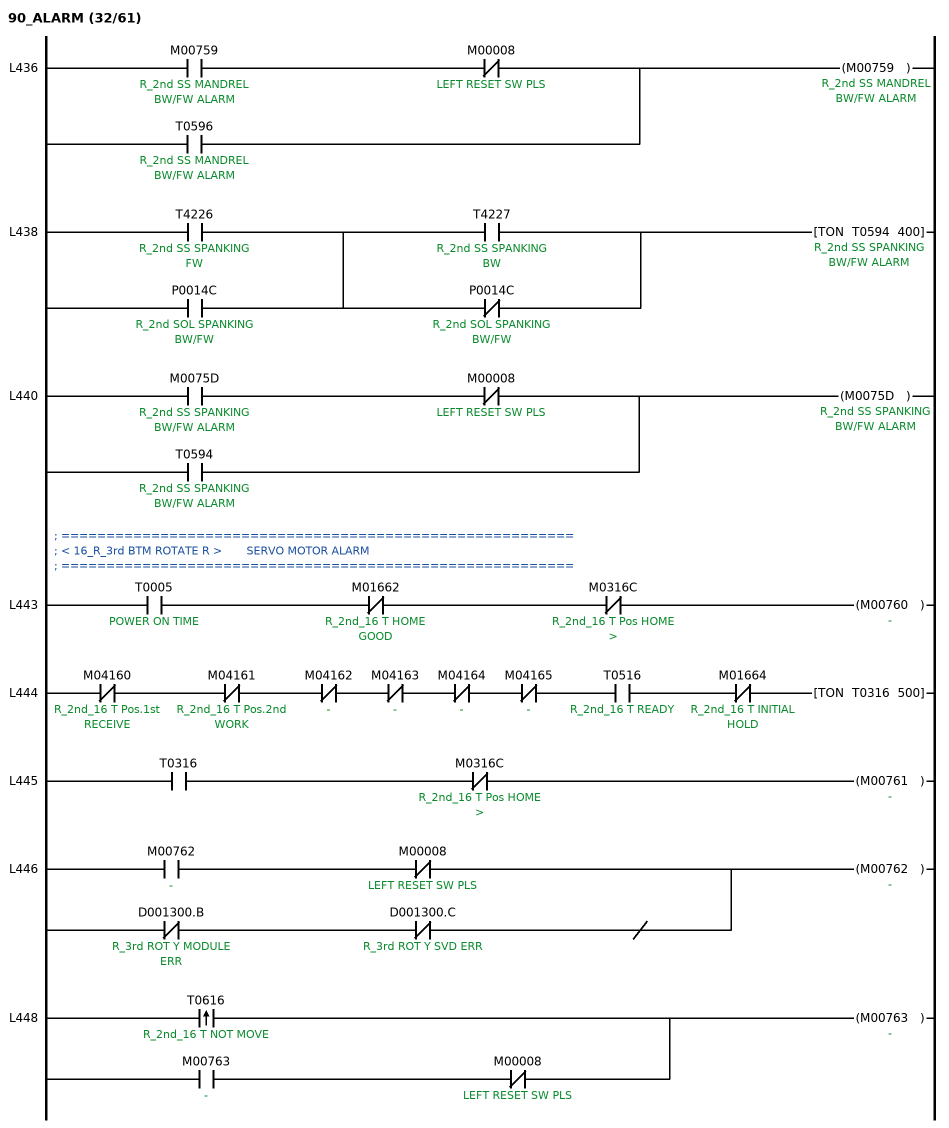
[picture p408: 90_ALARM rungs L436-L448]
; L436
LOAD      M00759	// R_2nd SS MANDREL BW/FW ALARM
AND NOT   M00008	// LEFT RESET SW PLS
OR        T0596	// R_2nd SS MANDREL BW/FW ALARM
OUT       M00759	// R_2nd SS MANDREL BW/FW ALARM
; L438
LOAD      T4226	// R_2nd SS SPANKING FW
OR        P0014C	// R_2nd SOL SPANKING BW/FW
LOAD      T4227	// R_2nd SS SPANKING BW
OR NOT    P0014C	// R_2nd SOL SPANKING BW/FW
AND LOAD
TON       T0594 400	// R_2nd SS SPANKING BW/FW ALARM
; L440
LOAD      M0075D	// R_2nd SS SPANKING BW/FW ALARM
AND NOT   M00008	// LEFT RESET SW PLS
OR        T0594	// R_2nd SS SPANKING BW/FW ALARM
OUT       M0075D	// R_2nd SS SPANKING BW/FW ALARM
// =========================================================
// 
//        < 16_R_3rd BTM ROTATE R >       SERVO MOTOR ALARM
// 
// =========================================================
; L443
LOAD      T0005	// POWER ON TIME
AND NOT   M01662	// R_2nd_16 T HOME GOOD
AND NOT   M0316C	// R_2nd_16 T Pos HOME >
OUT       M00760	// -
; L444
LOAD NOT  M04160	// R_2nd_16 T Pos.1st RECEIVE
AND NOT   M04161	// R_2nd_16 T Pos.2nd WORK
AND NOT   M04162	// -
AND NOT   M04163	// -
AND NOT   M04164	// -
AND NOT   M04165	// -
AND       T0516	// R_2nd_16 T READY
AND NOT   M01664	// R_2nd_16 T INITIAL HOLD
TON       T0316 500
; L445
LOAD      T0316
AND NOT   M0316C	// R_2nd_16 T Pos HOME >
OUT       M00761	// -
; L446
LOAD      M00762	// -
AND NOT   M00008	// LEFT RESET SW PLS
LOAD NOT  D001300.B	// R_3rd ROT Y MODULE ERR
AND NOT   D001300.C	// R_3rd ROT Y SVD ERR
NOT
OR LOAD
OUT       M00762	// -
; L448
LOADP     T0616	// R_2nd_16 T NOT MOVE
LOAD      M00763	// -
AND NOT   M00008	// LEFT RESET SW PLS
OR LOAD
OUT       M00763	// -

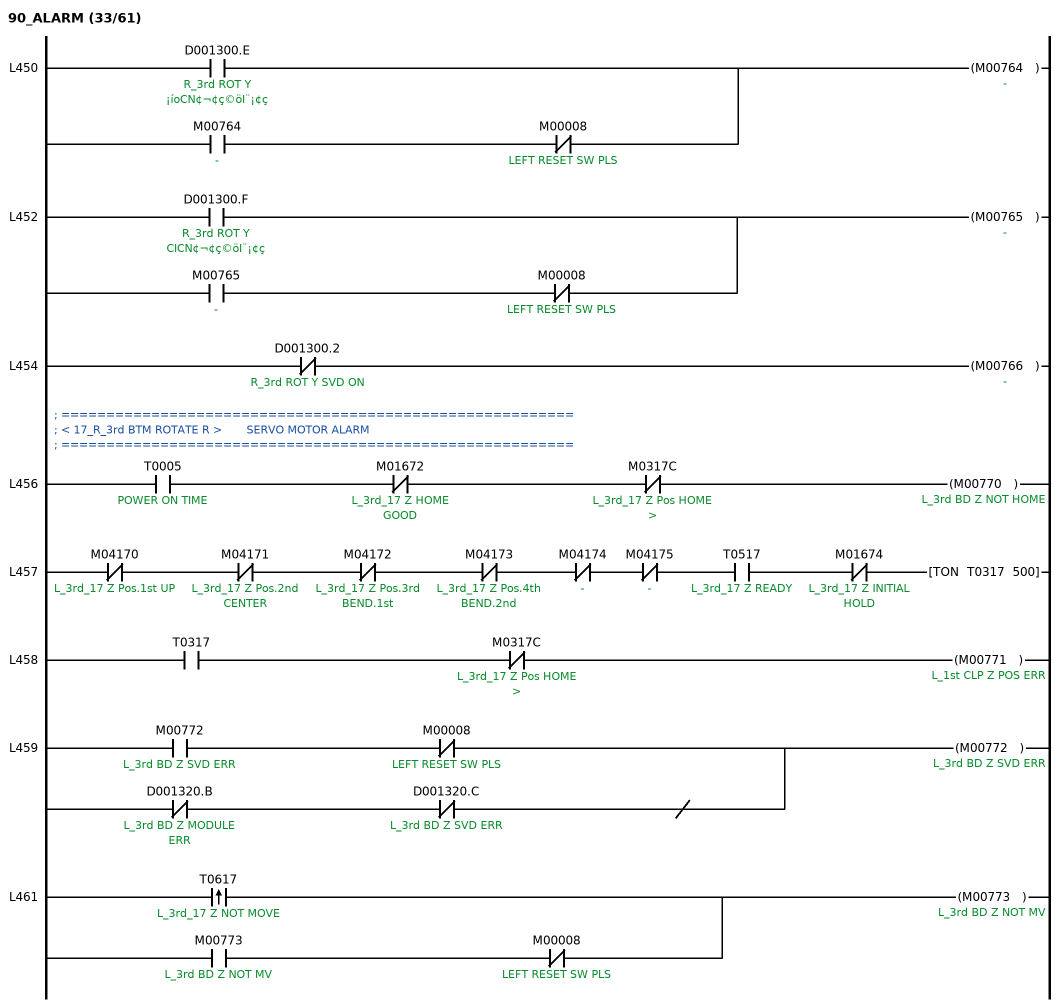
; L450
LOAD      D001300.E	// R_3rd ROT Y ¡íoCN¢¬¢ç©öI¨¡¢ç
LOAD      M00764	// -
AND NOT   M00008	// LEFT RESET SW PLS
OR LOAD
OUT       M00764	// -
; L452
LOAD      D001300.F	// R_3rd ROT Y CICN¢¬¢ç©öI¨¡¢ç
LOAD      M00765	// -
AND NOT   M00008	// LEFT RESET SW PLS
OR LOAD
OUT       M00765	// -
; L454
LOAD NOT  D001300.2	// R_3rd ROT Y SVD ON
OUT       M00766	// -
// =========================================================
// 
//        < 17_R_3rd BTM ROTATE R >       SERVO MOTOR ALARM
// 
// =========================================================
; L456
LOAD      T0005	// POWER ON TIME
AND NOT   M01672	// L_3rd_17 Z HOME GOOD
AND NOT   M0317C	// L_3rd_17 Z Pos HOME >
OUT       M00770	// L_3rd BD Z NOT HOME
; L457
LOAD NOT  M04170	// L_3rd_17 Z Pos.1st UP
AND NOT   M04171	// L_3rd_17 Z Pos.2nd CENTER
AND NOT   M04172	// L_3rd_17 Z Pos.3rd BEND.1st
AND NOT   M04173	// L_3rd_17 Z Pos.4th BEND.2nd
AND NOT   M04174	// -
AND NOT   M04175	// -
AND       T0517	// L_3rd_17 Z READY
AND NOT   M01674	// L_3rd_17 Z INITIAL HOLD
TON       T0317 500
; L458
LOAD      T0317
AND NOT   M0317C	// L_3rd_17 Z Pos HOME >
OUT       M00771	// L_1st CLP Z POS ERR
; L459
LOAD      M00772	// L_3rd BD Z SVD ERR
AND NOT   M00008	// LEFT RESET SW PLS
LOAD NOT  D001320.B	// L_3rd BD Z MODULE ERR
AND NOT   D001320.C	// L_3rd BD Z SVD ERR
NOT
OR LOAD
OUT       M00772	// L_3rd BD Z SVD ERR
; L461
LOADP     T0617	// L_3rd_17 Z NOT MOVE
LOAD      M00773	// L_3rd BD Z NOT MV
AND NOT   M00008	// LEFT RESET SW PLS
OR LOAD
OUT       M00773	// L_3rd BD Z NOT MV

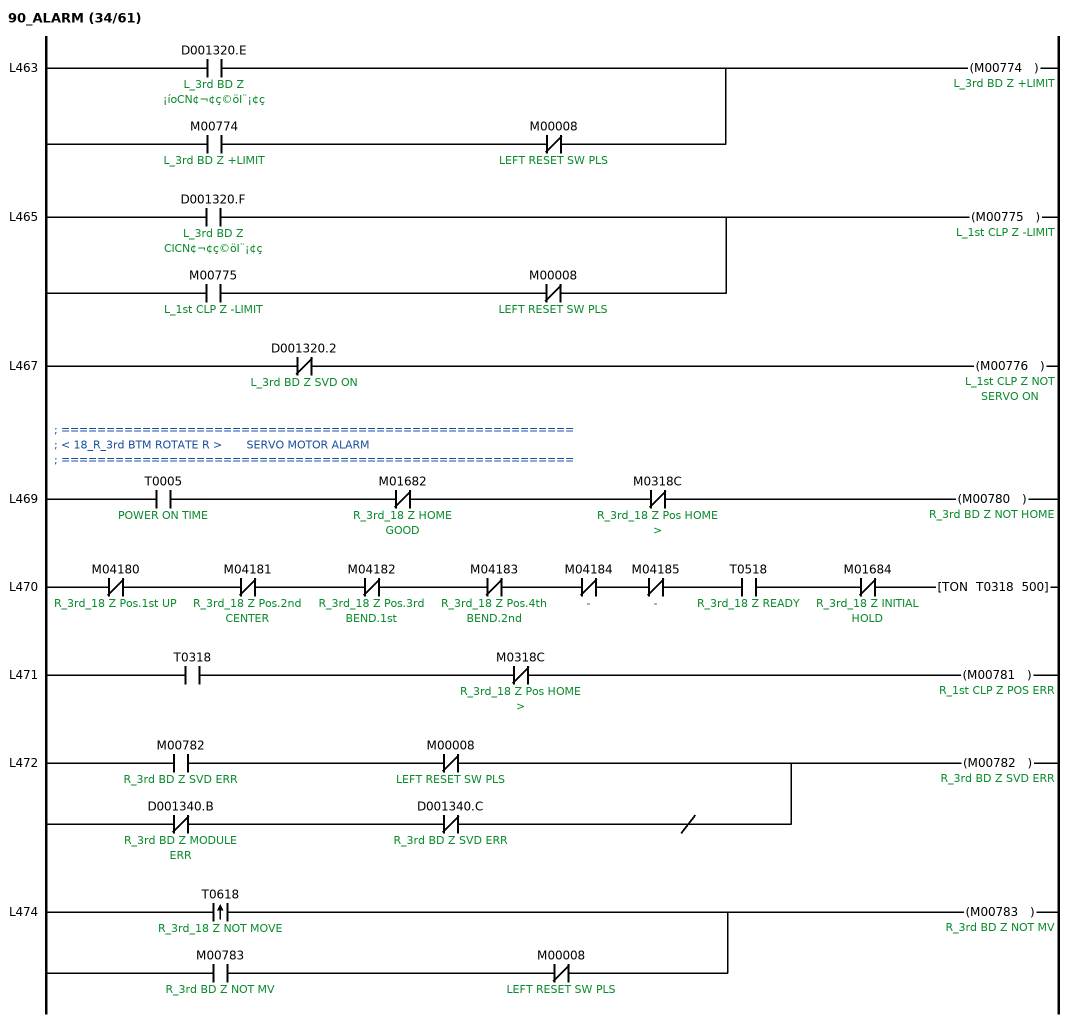
; L463
LOAD      D001320.E	// L_3rd BD Z ¡íoCN¢¬¢ç©öI¨¡¢ç
LOAD      M00774	// L_3rd BD Z +LIMIT
AND NOT   M00008	// LEFT RESET SW PLS
OR LOAD
OUT       M00774	// L_3rd BD Z +LIMIT
; L465
LOAD      D001320.F	// L_3rd BD Z CICN¢¬¢ç©öI¨¡¢ç
LOAD      M00775	// L_1st CLP Z -LIMIT
AND NOT   M00008	// LEFT RESET SW PLS
OR LOAD
OUT       M00775	// L_1st CLP Z -LIMIT
; L467
LOAD NOT  D001320.2	// L_3rd BD Z SVD ON
OUT       M00776	// L_1st CLP Z NOT SERVO ON
// =========================================================
// 
//        < 18_R_3rd BTM ROTATE R >       SERVO MOTOR ALARM
// 
// =========================================================
; L469
LOAD      T0005	// POWER ON TIME
AND NOT   M01682	// R_3rd_18 Z HOME GOOD
AND NOT   M0318C	// R_3rd_18 Z Pos HOME >
OUT       M00780	// R_3rd BD Z NOT HOME
; L470
LOAD NOT  M04180	// R_3rd_18 Z Pos.1st UP
AND NOT   M04181	// R_3rd_18 Z Pos.2nd CENTER
AND NOT   M04182	// R_3rd_18 Z Pos.3rd BEND.1st
AND NOT   M04183	// R_3rd_18 Z Pos.4th BEND.2nd
AND NOT   M04184	// -
AND NOT   M04185	// -
AND       T0518	// R_3rd_18 Z READY
AND NOT   M01684	// R_3rd_18 Z INITIAL HOLD
TON       T0318 500
; L471
LOAD      T0318
AND NOT   M0318C	// R_3rd_18 Z Pos HOME >
OUT       M00781	// R_1st CLP Z POS ERR
; L472
LOAD      M00782	// R_3rd BD Z SVD ERR
AND NOT   M00008	// LEFT RESET SW PLS
LOAD NOT  D001340.B	// R_3rd BD Z MODULE ERR
AND NOT   D001340.C	// R_3rd BD Z SVD ERR
NOT
OR LOAD
OUT       M00782	// R_3rd BD Z SVD ERR
; L474
LOADP     T0618	// R_3rd_18 Z NOT MOVE
LOAD      M00783	// R_3rd BD Z NOT MV
AND NOT   M00008	// LEFT RESET SW PLS
OR LOAD
OUT       M00783	// R_3rd BD Z NOT MV

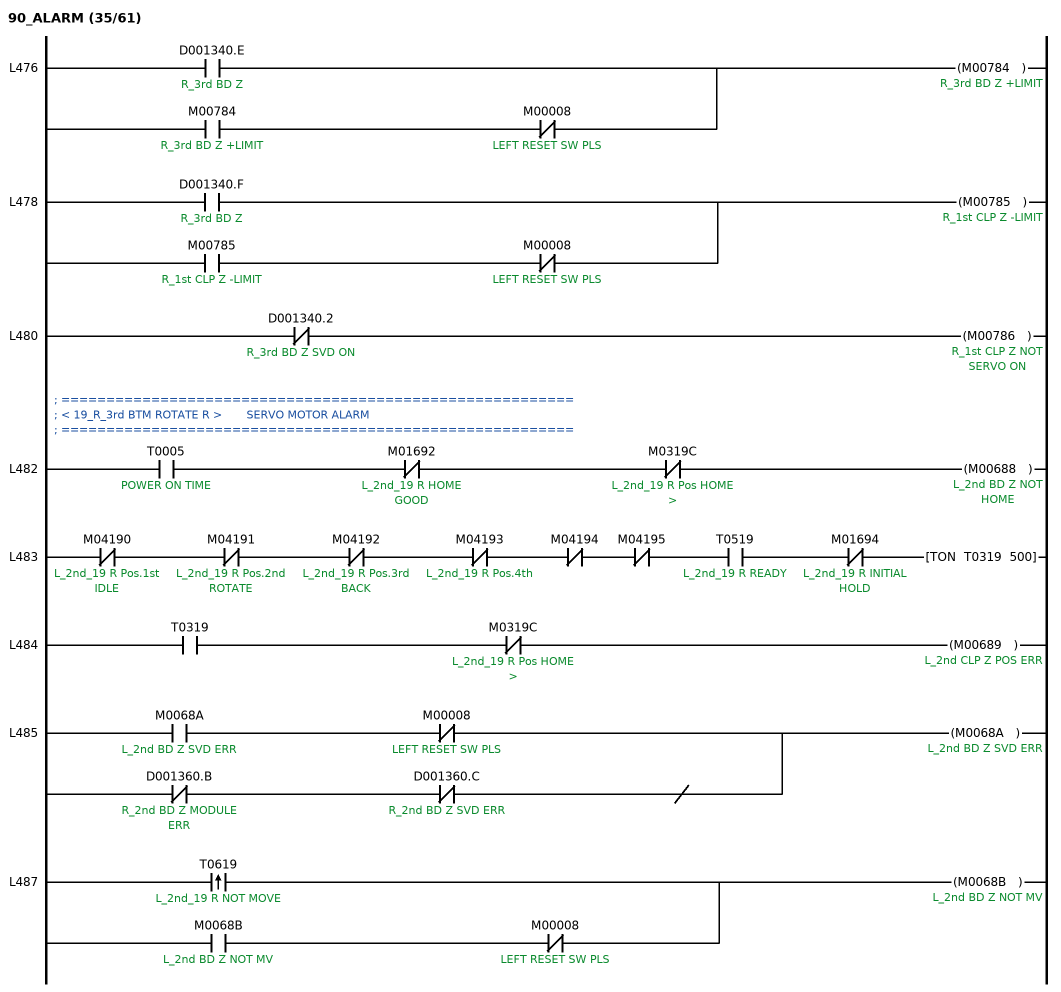
; L476
LOAD      D001340.E	// R_3rd BD Z
LOAD      M00784	// R_3rd BD Z +LIMIT
AND NOT   M00008	// LEFT RESET SW PLS
OR LOAD
OUT       M00784	// R_3rd BD Z +LIMIT
; L478
LOAD      D001340.F	// R_3rd BD Z
LOAD      M00785	// R_1st CLP Z -LIMIT
AND NOT   M00008	// LEFT RESET SW PLS
OR LOAD
OUT       M00785	// R_1st CLP Z -LIMIT
; L480
LOAD NOT  D001340.2	// R_3rd BD Z SVD ON
OUT       M00786	// R_1st CLP Z NOT SERVO ON
// =========================================================
// 
//        < 19_R_3rd BTM ROTATE R >       SERVO MOTOR ALARM
// 
// =========================================================
; L482
LOAD      T0005	// POWER ON TIME
AND NOT   M01692	// L_2nd_19 R HOME GOOD
AND NOT   M0319C	// L_2nd_19 R Pos HOME >
OUT       M00688	// L_2nd BD Z NOT HOME
; L483
LOAD NOT  M04190	// L_2nd_19 R Pos.1st IDLE
AND NOT   M04191	// L_2nd_19 R Pos.2nd ROTATE
AND NOT   M04192	// L_2nd_19 R Pos.3rd BACK
AND NOT   M04193	// L_2nd_19 R Pos.4th 
AND NOT   M04194
AND NOT   M04195
AND       T0519	// L_2nd_19 R READY
AND NOT   M01694	// L_2nd_19 R INITIAL HOLD
TON       T0319 500
; L484
LOAD      T0319
AND NOT   M0319C	// L_2nd_19 R Pos HOME >
OUT       M00689	// L_2nd CLP Z POS ERR
; L485
LOAD      M0068A	// L_2nd BD Z SVD ERR
AND NOT   M00008	// LEFT RESET SW PLS
LOAD NOT  D001360.B	// R_2nd BD Z MODULE ERR
AND NOT   D001360.C	// R_2nd BD Z SVD ERR
NOT
OR LOAD
OUT       M0068A	// L_2nd BD Z SVD ERR
; L487
LOADP     T0619	// L_2nd_19 R NOT MOVE
LOAD      M0068B	// L_2nd BD Z NOT MV
AND NOT   M00008	// LEFT RESET SW PLS
OR LOAD
OUT       M0068B	// L_2nd BD Z NOT MV

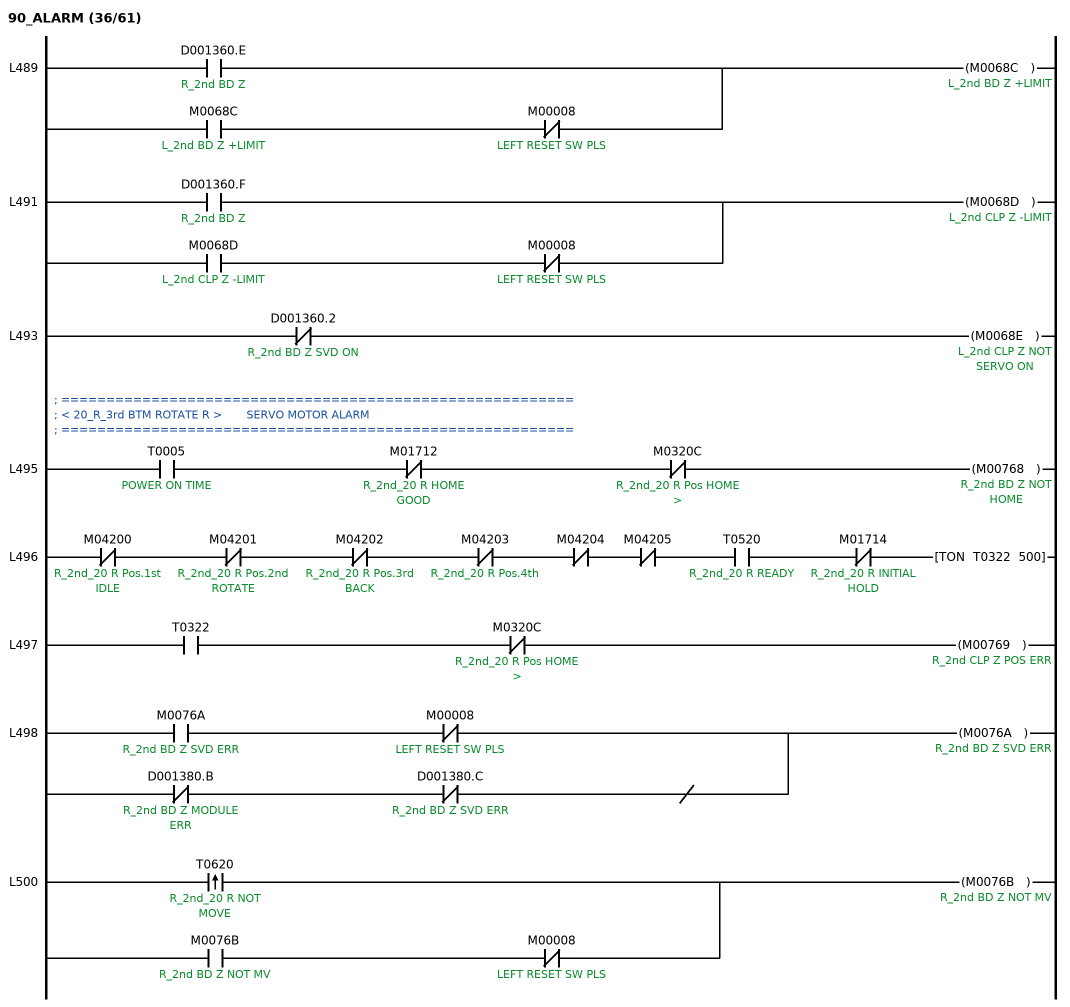
; L489
LOAD      D001360.E	// R_2nd BD Z
LOAD      M0068C	// L_2nd BD Z +LIMIT
AND NOT   M00008	// LEFT RESET SW PLS
OR LOAD
OUT       M0068C	// L_2nd BD Z +LIMIT
; L491
LOAD      D001360.F	// R_2nd BD Z
LOAD      M0068D	// L_2nd CLP Z -LIMIT
AND NOT   M00008	// LEFT RESET SW PLS
OR LOAD
OUT       M0068D	// L_2nd CLP Z -LIMIT
; L493
LOAD NOT  D001360.2	// R_2nd BD Z SVD ON
OUT       M0068E	// L_2nd CLP Z NOT SERVO ON
// =========================================================
// 
//        < 20_R_3rd BTM ROTATE R >       SERVO MOTOR ALARM
// 
// =========================================================
; L495
LOAD      T0005	// POWER ON TIME
AND NOT   M01712	// R_2nd_20 R HOME GOOD
AND NOT   M0320C	// R_2nd_20 R Pos HOME >
OUT       M00768	// R_2nd BD Z NOT HOME
; L496
LOAD NOT  M04200	// R_2nd_20 R Pos.1st IDLE
AND NOT   M04201	// R_2nd_20 R Pos.2nd ROTATE
AND NOT   M04202	// R_2nd_20 R Pos.3rd BACK
AND NOT   M04203	// R_2nd_20 R Pos.4th 
AND NOT   M04204
AND NOT   M04205
AND       T0520	// R_2nd_20 R READY
AND NOT   M01714	// R_2nd_20 R INITIAL HOLD
TON       T0322 500
; L497
LOAD      T0322
AND NOT   M0320C	// R_2nd_20 R Pos HOME >
OUT       M00769	// R_2nd CLP Z POS ERR
; L498
LOAD      M0076A	// R_2nd BD Z SVD ERR
AND NOT   M00008	// LEFT RESET SW PLS
LOAD NOT  D001380.B	// R_2nd BD Z MODULE ERR
AND NOT   D001380.C	// R_2nd BD Z SVD ERR
NOT
OR LOAD
OUT       M0076A	// R_2nd BD Z SVD ERR
; L500
LOADP     T0620	// R_2nd_20 R NOT MOVE
LOAD      M0076B	// R_2nd BD Z NOT MV
AND NOT   M00008	// LEFT RESET SW PLS
OR LOAD
OUT       M0076B	// R_2nd BD Z NOT MV

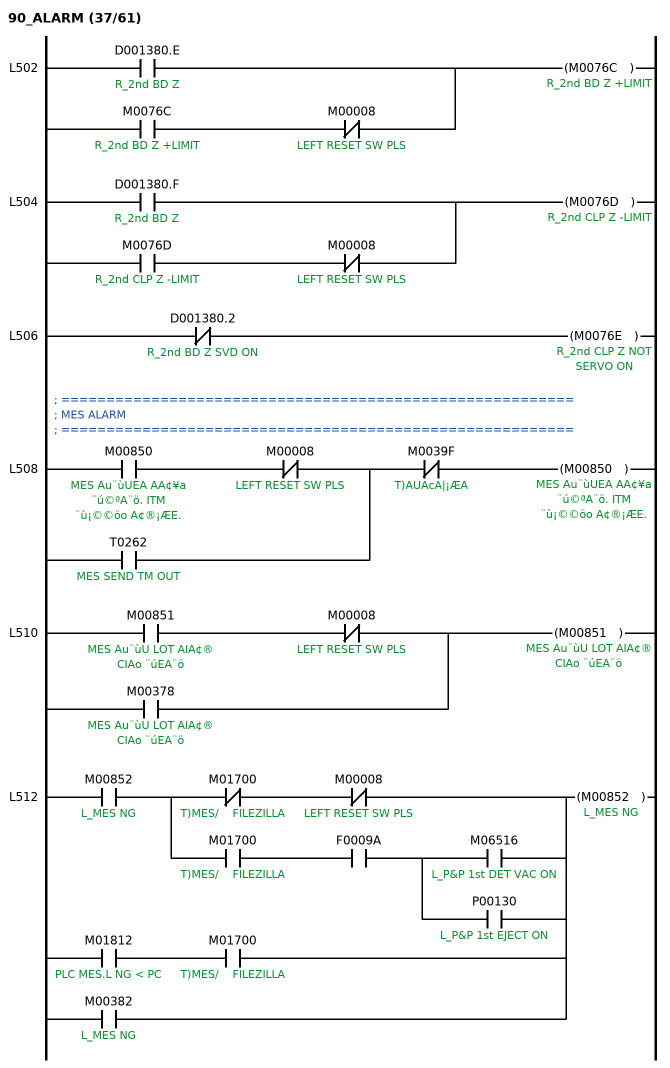
; L502
LOAD      D001380.E	// R_2nd BD Z
LOAD      M0076C	// R_2nd BD Z +LIMIT
AND NOT   M00008	// LEFT RESET SW PLS
OR LOAD
OUT       M0076C	// R_2nd BD Z +LIMIT
; L504
LOAD      D001380.F	// R_2nd BD Z
LOAD      M0076D	// R_2nd CLP Z -LIMIT
AND NOT   M00008	// LEFT RESET SW PLS
OR LOAD
OUT       M0076D	// R_2nd CLP Z -LIMIT
; L506
LOAD NOT  D001380.2	// R_2nd BD Z SVD ON
OUT       M0076E	// R_2nd CLP Z NOT SERVO ON
// =========================================================
// 
//        MES ALARM
// 
// =========================================================
; L508
LOAD      M00850	// MES Au¨ùUEA AA¢¥a ¨ú©ªA¨ö. ITM ¨ù¡©©öo A¢®¡ÆE.
AND NOT   M00008	// LEFT RESET SW PLS
OR        T0262	// MES SEND TM OUT
AND NOT   M0039F	// T)AUAcA|¡ÆA
OUT       M00850	// MES Au¨ùUEA AA¢¥a ¨ú©ªA¨ö. ITM ¨ù¡©©öo A¢®¡ÆE.
; L510
LOAD      M00851	// MES Au¨ùU LOT AIA¢® CIAo ¨úEA¨ö
AND NOT   M00008	// LEFT RESET SW PLS
OR        M00378	// MES Au¨ùU LOT AIA¢® CIAo ¨úEA¨ö
OUT       M00851	// MES Au¨ùU LOT AIA¢® CIAo ¨úEA¨ö
; L512
LOAD      M00852	// L_MES NG
LOAD NOT  M01700	// T)MES/    FILEZILLA
AND NOT   M00008	// LEFT RESET SW PLS
LOAD      M01700	// T)MES/    FILEZILLA
AND       F0009A
LOAD      M06516	// L_P&P 1st DET VAC ON
OR        P00130	// L_P&P 1st EJECT ON
AND LOAD
OR LOAD
AND LOAD
LOAD      M01812	// PLC MES.L NG < PC
AND       M01700	// T)MES/    FILEZILLA
OR LOAD
OR        M00382	// L_MES NG
OUT       M00852	// L_MES NG

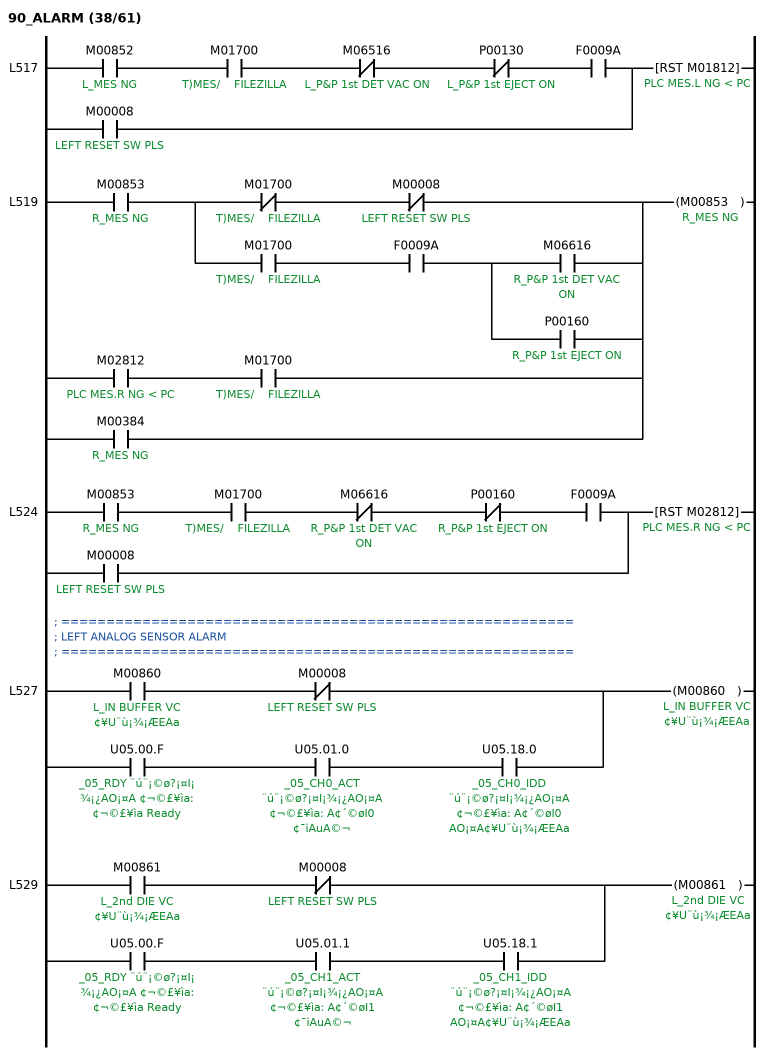
; L517
LOAD      M00852	// L_MES NG
AND       M01700	// T)MES/    FILEZILLA
AND NOT   M06516	// L_P&P 1st DET VAC ON
AND NOT   P00130	// L_P&P 1st EJECT ON
AND       F0009A
OR        M00008	// LEFT RESET SW PLS
RST       M01812	// PLC MES.L NG < PC
; L519
LOAD      M00853	// R_MES NG
LOAD NOT  M01700	// T)MES/    FILEZILLA
AND NOT   M00008	// LEFT RESET SW PLS
LOAD      M01700	// T)MES/    FILEZILLA
AND       F0009A
LOAD      M06616	// R_P&P 1st DET VAC ON
OR        P00160	// R_P&P 1st EJECT ON
AND LOAD
OR LOAD
AND LOAD
LOAD      M02812	// PLC MES.R NG < PC
AND       M01700	// T)MES/    FILEZILLA
OR LOAD
OR        M00384	// R_MES NG
OUT       M00853	// R_MES NG
; L524
LOAD      M00853	// R_MES NG
AND       M01700	// T)MES/    FILEZILLA
AND NOT   M06616	// R_P&P 1st DET VAC ON
AND NOT   P00160	// R_P&P 1st EJECT ON
AND       F0009A
OR        M00008	// LEFT RESET SW PLS
RST       M02812	// PLC MES.R NG < PC
// =========================================================
// 
//        LEFT ANALOG SENSOR ALARM
// 
// =========================================================
; L527
LOAD      M00860	// L_IN BUFFER VC ¢¥U¨ù¡¾¡ÆEAa
AND NOT   M00008	// LEFT RESET SW PLS
LOAD      U05.00.F	// _05_RDY ¨ú¨¡©ø?¡¤I¡¾¡¿AO¡¤A ¢¬©£¥ìa: ¢¬©£¥ìa Ready
AND       U05.01.0	// _05_CH0_ACT ¨ú¨¡©ø?¡¤I¡¾¡¿AO¡¤A ¢¬©£¥ìa: A¢´©øI0 ¢¯iAuA©¬
AND       U05.18.0	// _05_CH0_IDD ¨ú¨¡©ø?¡¤I¡¾¡¿AO¡¤A ¢¬©£¥ìa: A¢´©øI0 AO¡¤A¢¥U¨ù¡¾¡ÆEAa
OR LOAD
OUT       M00860	// L_IN BUFFER VC ¢¥U¨ù¡¾¡ÆEAa
; L529
LOAD      M00861	// L_2nd DIE VC ¢¥U¨ù¡¾¡ÆEAa
AND NOT   M00008	// LEFT RESET SW PLS
LOAD      U05.00.F	// _05_RDY ¨ú¨¡©ø?¡¤I¡¾¡¿AO¡¤A ¢¬©£¥ìa: ¢¬©£¥ìa Ready
AND       U05.01.1	// _05_CH1_ACT ¨ú¨¡©ø?¡¤I¡¾¡¿AO¡¤A ¢¬©£¥ìa: A¢´©øI1 ¢¯iAuA©¬
AND       U05.18.1	// _05_CH1_IDD ¨ú¨¡©ø?¡¤I¡¾¡¿AO¡¤A ¢¬©£¥ìa: A¢´©øI1 AO¡¤A¢¥U¨ù¡¾¡ÆEAa
OR LOAD
OUT       M00861	// L_2nd DIE VC ¢¥U¨ù¡¾¡ÆEAa

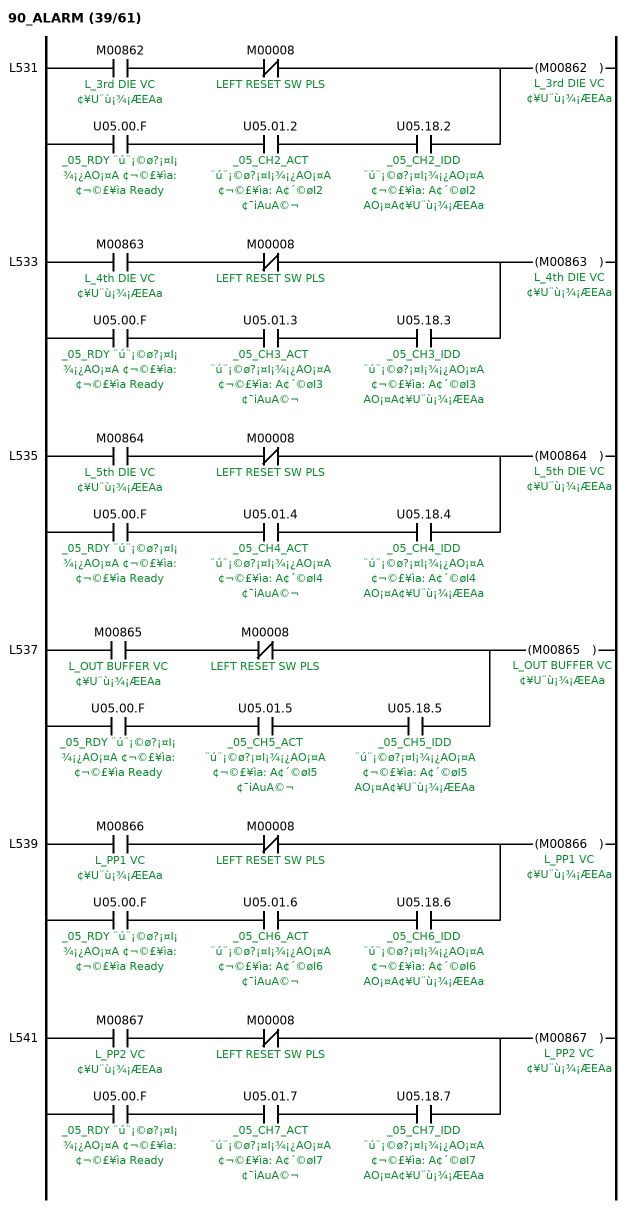
; L531
LOAD      M00862	// L_3rd DIE VC ¢¥U¨ù¡¾¡ÆEAa
AND NOT   M00008	// LEFT RESET SW PLS
LOAD      U05.00.F	// _05_RDY ¨ú¨¡©ø?¡¤I¡¾¡¿AO¡¤A ¢¬©£¥ìa: ¢¬©£¥ìa Ready
AND       U05.01.2	// _05_CH2_ACT ¨ú¨¡©ø?¡¤I¡¾¡¿AO¡¤A ¢¬©£¥ìa: A¢´©øI2 ¢¯iAuA©¬
AND       U05.18.2	// _05_CH2_IDD ¨ú¨¡©ø?¡¤I¡¾¡¿AO¡¤A ¢¬©£¥ìa: A¢´©øI2 AO¡¤A¢¥U¨ù¡¾¡ÆEAa
OR LOAD
OUT       M00862	// L_3rd DIE VC ¢¥U¨ù¡¾¡ÆEAa
; L533
LOAD      M00863	// L_4th DIE VC ¢¥U¨ù¡¾¡ÆEAa
AND NOT   M00008	// LEFT RESET SW PLS
LOAD      U05.00.F	// _05_RDY ¨ú¨¡©ø?¡¤I¡¾¡¿AO¡¤A ¢¬©£¥ìa: ¢¬©£¥ìa Ready
AND       U05.01.3	// _05_CH3_ACT ¨ú¨¡©ø?¡¤I¡¾¡¿AO¡¤A ¢¬©£¥ìa: A¢´©øI3 ¢¯iAuA©¬
AND       U05.18.3	// _05_CH3_IDD ¨ú¨¡©ø?¡¤I¡¾¡¿AO¡¤A ¢¬©£¥ìa: A¢´©øI3 AO¡¤A¢¥U¨ù¡¾¡ÆEAa
OR LOAD
OUT       M00863	// L_4th DIE VC ¢¥U¨ù¡¾¡ÆEAa
; L535
LOAD      M00864	// L_5th DIE VC ¢¥U¨ù¡¾¡ÆEAa
AND NOT   M00008	// LEFT RESET SW PLS
LOAD      U05.00.F	// _05_RDY ¨ú¨¡©ø?¡¤I¡¾¡¿AO¡¤A ¢¬©£¥ìa: ¢¬©£¥ìa Ready
AND       U05.01.4	// _05_CH4_ACT ¨ú¨¡©ø?¡¤I¡¾¡¿AO¡¤A ¢¬©£¥ìa: A¢´©øI4 ¢¯iAuA©¬
AND       U05.18.4	// _05_CH4_IDD ¨ú¨¡©ø?¡¤I¡¾¡¿AO¡¤A ¢¬©£¥ìa: A¢´©øI4 AO¡¤A¢¥U¨ù¡¾¡ÆEAa
OR LOAD
OUT       M00864	// L_5th DIE VC ¢¥U¨ù¡¾¡ÆEAa
; L537
LOAD      M00865	// L_OUT BUFFER VC ¢¥U¨ù¡¾¡ÆEAa
AND NOT   M00008	// LEFT RESET SW PLS
LOAD      U05.00.F	// _05_RDY ¨ú¨¡©ø?¡¤I¡¾¡¿AO¡¤A ¢¬©£¥ìa: ¢¬©£¥ìa Ready
AND       U05.01.5	// _05_CH5_ACT ¨ú¨¡©ø?¡¤I¡¾¡¿AO¡¤A ¢¬©£¥ìa: A¢´©øI5 ¢¯iAuA©¬
AND       U05.18.5	// _05_CH5_IDD ¨ú¨¡©ø?¡¤I¡¾¡¿AO¡¤A ¢¬©£¥ìa: A¢´©øI5 AO¡¤A¢¥U¨ù¡¾¡ÆEAa
OR LOAD
OUT       M00865	// L_OUT BUFFER VC ¢¥U¨ù¡¾¡ÆEAa
; L539
LOAD      M00866	// L_PP1 VC ¢¥U¨ù¡¾¡ÆEAa
AND NOT   M00008	// LEFT RESET SW PLS
LOAD      U05.00.F	// _05_RDY ¨ú¨¡©ø?¡¤I¡¾¡¿AO¡¤A ¢¬©£¥ìa: ¢¬©£¥ìa Ready
AND       U05.01.6	// _05_CH6_ACT ¨ú¨¡©ø?¡¤I¡¾¡¿AO¡¤A ¢¬©£¥ìa: A¢´©øI6 ¢¯iAuA©¬
AND       U05.18.6	// _05_CH6_IDD ¨ú¨¡©ø?¡¤I¡¾¡¿AO¡¤A ¢¬©£¥ìa: A¢´©øI6 AO¡¤A¢¥U¨ù¡¾¡ÆEAa
OR LOAD
OUT       M00866	// L_PP1 VC ¢¥U¨ù¡¾¡ÆEAa
; L541
LOAD      M00867	// L_PP2 VC ¢¥U¨ù¡¾¡ÆEAa
AND NOT   M00008	// LEFT RESET SW PLS
LOAD      U05.00.F	// _05_RDY ¨ú¨¡©ø?¡¤I¡¾¡¿AO¡¤A ¢¬©£¥ìa: ¢¬©£¥ìa Ready
AND       U05.01.7	// _05_CH7_ACT ¨ú¨¡©ø?¡¤I¡¾¡¿AO¡¤A ¢¬©£¥ìa: A¢´©øI7 ¢¯iAuA©¬
AND       U05.18.7	// _05_CH7_IDD ¨ú¨¡©ø?¡¤I¡¾¡¿AO¡¤A ¢¬©£¥ìa: A¢´©øI7 AO¡¤A¢¥U¨ù¡¾¡ÆEAa
OR LOAD
OUT       M00867	// L_PP2 VC ¢¥U¨ù¡¾¡ÆEAa

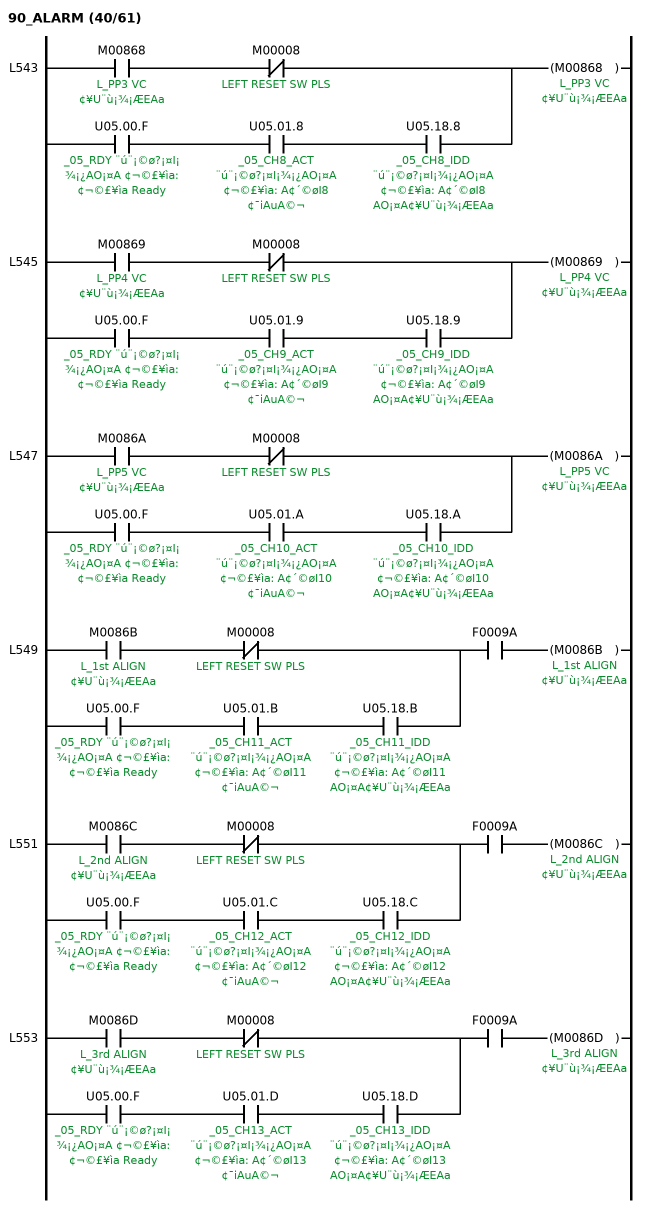
; L543
LOAD      M00868	// L_PP3 VC ¢¥U¨ù¡¾¡ÆEAa
AND NOT   M00008	// LEFT RESET SW PLS
LOAD      U05.00.F	// _05_RDY ¨ú¨¡©ø?¡¤I¡¾¡¿AO¡¤A ¢¬©£¥ìa: ¢¬©£¥ìa Ready
AND       U05.01.8	// _05_CH8_ACT ¨ú¨¡©ø?¡¤I¡¾¡¿AO¡¤A ¢¬©£¥ìa: A¢´©øI8 ¢¯iAuA©¬
AND       U05.18.8	// _05_CH8_IDD ¨ú¨¡©ø?¡¤I¡¾¡¿AO¡¤A ¢¬©£¥ìa: A¢´©øI8 AO¡¤A¢¥U¨ù¡¾¡ÆEAa
OR LOAD
OUT       M00868	// L_PP3 VC ¢¥U¨ù¡¾¡ÆEAa
; L545
LOAD      M00869	// L_PP4 VC ¢¥U¨ù¡¾¡ÆEAa
AND NOT   M00008	// LEFT RESET SW PLS
LOAD      U05.00.F	// _05_RDY ¨ú¨¡©ø?¡¤I¡¾¡¿AO¡¤A ¢¬©£¥ìa: ¢¬©£¥ìa Ready
AND       U05.01.9	// _05_CH9_ACT ¨ú¨¡©ø?¡¤I¡¾¡¿AO¡¤A ¢¬©£¥ìa: A¢´©øI9 ¢¯iAuA©¬
AND       U05.18.9	// _05_CH9_IDD ¨ú¨¡©ø?¡¤I¡¾¡¿AO¡¤A ¢¬©£¥ìa: A¢´©øI9 AO¡¤A¢¥U¨ù¡¾¡ÆEAa
OR LOAD
OUT       M00869	// L_PP4 VC ¢¥U¨ù¡¾¡ÆEAa
; L547
LOAD      M0086A	// L_PP5 VC ¢¥U¨ù¡¾¡ÆEAa
AND NOT   M00008	// LEFT RESET SW PLS
LOAD      U05.00.F	// _05_RDY ¨ú¨¡©ø?¡¤I¡¾¡¿AO¡¤A ¢¬©£¥ìa: ¢¬©£¥ìa Ready
AND       U05.01.A	// _05_CH10_ACT ¨ú¨¡©ø?¡¤I¡¾¡¿AO¡¤A ¢¬©£¥ìa: A¢´©øI10 ¢¯iAuA©¬
AND       U05.18.A	// _05_CH10_IDD ¨ú¨¡©ø?¡¤I¡¾¡¿AO¡¤A ¢¬©£¥ìa: A¢´©øI10 AO¡¤A¢¥U¨ù¡¾¡ÆEAa
OR LOAD
OUT       M0086A	// L_PP5 VC ¢¥U¨ù¡¾¡ÆEAa
; L549
LOAD      M0086B	// L_1st ALIGN ¢¥U¨ù¡¾¡ÆEAa
AND NOT   M00008	// LEFT RESET SW PLS
LOAD      U05.00.F	// _05_RDY ¨ú¨¡©ø?¡¤I¡¾¡¿AO¡¤A ¢¬©£¥ìa: ¢¬©£¥ìa Ready
AND       U05.01.B	// _05_CH11_ACT ¨ú¨¡©ø?¡¤I¡¾¡¿AO¡¤A ¢¬©£¥ìa: A¢´©øI11 ¢¯iAuA©¬
AND       U05.18.B	// _05_CH11_IDD ¨ú¨¡©ø?¡¤I¡¾¡¿AO¡¤A ¢¬©£¥ìa: A¢´©øI11 AO¡¤A¢¥U¨ù¡¾¡ÆEAa
OR LOAD
AND       F0009A
OUT       M0086B	// L_1st ALIGN ¢¥U¨ù¡¾¡ÆEAa
; L551
LOAD      M0086C	// L_2nd ALIGN ¢¥U¨ù¡¾¡ÆEAa
AND NOT   M00008	// LEFT RESET SW PLS
LOAD      U05.00.F	// _05_RDY ¨ú¨¡©ø?¡¤I¡¾¡¿AO¡¤A ¢¬©£¥ìa: ¢¬©£¥ìa Ready
AND       U05.01.C	// _05_CH12_ACT ¨ú¨¡©ø?¡¤I¡¾¡¿AO¡¤A ¢¬©£¥ìa: A¢´©øI12 ¢¯iAuA©¬
AND       U05.18.C	// _05_CH12_IDD ¨ú¨¡©ø?¡¤I¡¾¡¿AO¡¤A ¢¬©£¥ìa: A¢´©øI12 AO¡¤A¢¥U¨ù¡¾¡ÆEAa
OR LOAD
AND       F0009A
OUT       M0086C	// L_2nd ALIGN ¢¥U¨ù¡¾¡ÆEAa
; L553
LOAD      M0086D	// L_3rd ALIGN ¢¥U¨ù¡¾¡ÆEAa
AND NOT   M00008	// LEFT RESET SW PLS
LOAD      U05.00.F	// _05_RDY ¨ú¨¡©ø?¡¤I¡¾¡¿AO¡¤A ¢¬©£¥ìa: ¢¬©£¥ìa Ready
AND       U05.01.D	// _05_CH13_ACT ¨ú¨¡©ø?¡¤I¡¾¡¿AO¡¤A ¢¬©£¥ìa: A¢´©øI13 ¢¯iAuA©¬
AND       U05.18.D	// _05_CH13_IDD ¨ú¨¡©ø?¡¤I¡¾¡¿AO¡¤A ¢¬©£¥ìa: A¢´©øI13 AO¡¤A¢¥U¨ù¡¾¡ÆEAa
OR LOAD
AND       F0009A
OUT       M0086D	// L_3rd ALIGN ¢¥U¨ù¡¾¡ÆEAa

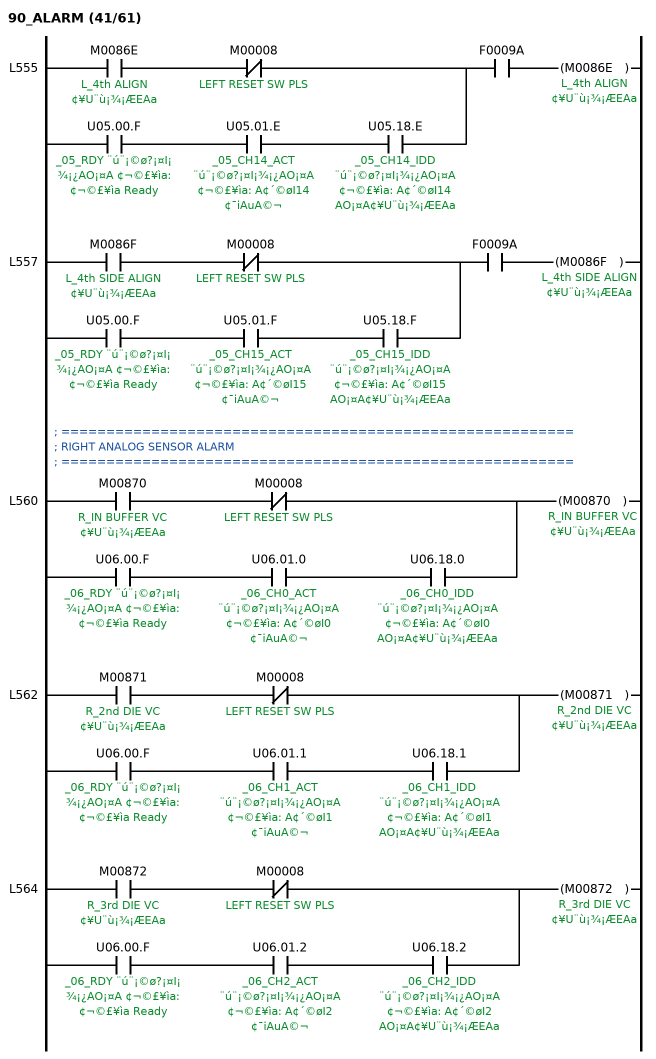
; L555
LOAD      M0086E	// L_4th ALIGN ¢¥U¨ù¡¾¡ÆEAa
AND NOT   M00008	// LEFT RESET SW PLS
LOAD      U05.00.F	// _05_RDY ¨ú¨¡©ø?¡¤I¡¾¡¿AO¡¤A ¢¬©£¥ìa: ¢¬©£¥ìa Ready
AND       U05.01.E	// _05_CH14_ACT ¨ú¨¡©ø?¡¤I¡¾¡¿AO¡¤A ¢¬©£¥ìa: A¢´©øI14 ¢¯iAuA©¬
AND       U05.18.E	// _05_CH14_IDD ¨ú¨¡©ø?¡¤I¡¾¡¿AO¡¤A ¢¬©£¥ìa: A¢´©øI14 AO¡¤A¢¥U¨ù¡¾¡ÆEAa
OR LOAD
AND       F0009A
OUT       M0086E	// L_4th ALIGN ¢¥U¨ù¡¾¡ÆEAa
; L557
LOAD      M0086F	// L_4th SIDE ALIGN ¢¥U¨ù¡¾¡ÆEAa
AND NOT   M00008	// LEFT RESET SW PLS
LOAD      U05.00.F	// _05_RDY ¨ú¨¡©ø?¡¤I¡¾¡¿AO¡¤A ¢¬©£¥ìa: ¢¬©£¥ìa Ready
AND       U05.01.F	// _05_CH15_ACT ¨ú¨¡©ø?¡¤I¡¾¡¿AO¡¤A ¢¬©£¥ìa: A¢´©øI15 ¢¯iAuA©¬
AND       U05.18.F	// _05_CH15_IDD ¨ú¨¡©ø?¡¤I¡¾¡¿AO¡¤A ¢¬©£¥ìa: A¢´©øI15 AO¡¤A¢¥U¨ù¡¾¡ÆEAa
OR LOAD
AND       F0009A
OUT       M0086F	// L_4th SIDE ALIGN ¢¥U¨ù¡¾¡ÆEAa
// =========================================================
// 
//        RIGHT ANALOG SENSOR ALARM
// 
// =========================================================
; L560
LOAD      M00870	// R_IN BUFFER VC ¢¥U¨ù¡¾¡ÆEAa
AND NOT   M00008	// LEFT RESET SW PLS
LOAD      U06.00.F	// _06_RDY ¨ú¨¡©ø?¡¤I¡¾¡¿AO¡¤A ¢¬©£¥ìa: ¢¬©£¥ìa Ready
AND       U06.01.0	// _06_CH0_ACT ¨ú¨¡©ø?¡¤I¡¾¡¿AO¡¤A ¢¬©£¥ìa: A¢´©øI0 ¢¯iAuA©¬
AND       U06.18.0	// _06_CH0_IDD ¨ú¨¡©ø?¡¤I¡¾¡¿AO¡¤A ¢¬©£¥ìa: A¢´©øI0 AO¡¤A¢¥U¨ù¡¾¡ÆEAa
OR LOAD
OUT       M00870	// R_IN BUFFER VC ¢¥U¨ù¡¾¡ÆEAa
; L562
LOAD      M00871	// R_2nd DIE VC ¢¥U¨ù¡¾¡ÆEAa
AND NOT   M00008	// LEFT RESET SW PLS
LOAD      U06.00.F	// _06_RDY ¨ú¨¡©ø?¡¤I¡¾¡¿AO¡¤A ¢¬©£¥ìa: ¢¬©£¥ìa Ready
AND       U06.01.1	// _06_CH1_ACT ¨ú¨¡©ø?¡¤I¡¾¡¿AO¡¤A ¢¬©£¥ìa: A¢´©øI1 ¢¯iAuA©¬
AND       U06.18.1	// _06_CH1_IDD ¨ú¨¡©ø?¡¤I¡¾¡¿AO¡¤A ¢¬©£¥ìa: A¢´©øI1 AO¡¤A¢¥U¨ù¡¾¡ÆEAa
OR LOAD
OUT       M00871	// R_2nd DIE VC ¢¥U¨ù¡¾¡ÆEAa
; L564
LOAD      M00872	// R_3rd DIE VC ¢¥U¨ù¡¾¡ÆEAa
AND NOT   M00008	// LEFT RESET SW PLS
LOAD      U06.00.F	// _06_RDY ¨ú¨¡©ø?¡¤I¡¾¡¿AO¡¤A ¢¬©£¥ìa: ¢¬©£¥ìa Ready
AND       U06.01.2	// _06_CH2_ACT ¨ú¨¡©ø?¡¤I¡¾¡¿AO¡¤A ¢¬©£¥ìa: A¢´©øI2 ¢¯iAuA©¬
AND       U06.18.2	// _06_CH2_IDD ¨ú¨¡©ø?¡¤I¡¾¡¿AO¡¤A ¢¬©£¥ìa: A¢´©øI2 AO¡¤A¢¥U¨ù¡¾¡ÆEAa
OR LOAD
OUT       M00872	// R_3rd DIE VC ¢¥U¨ù¡¾¡ÆEAa

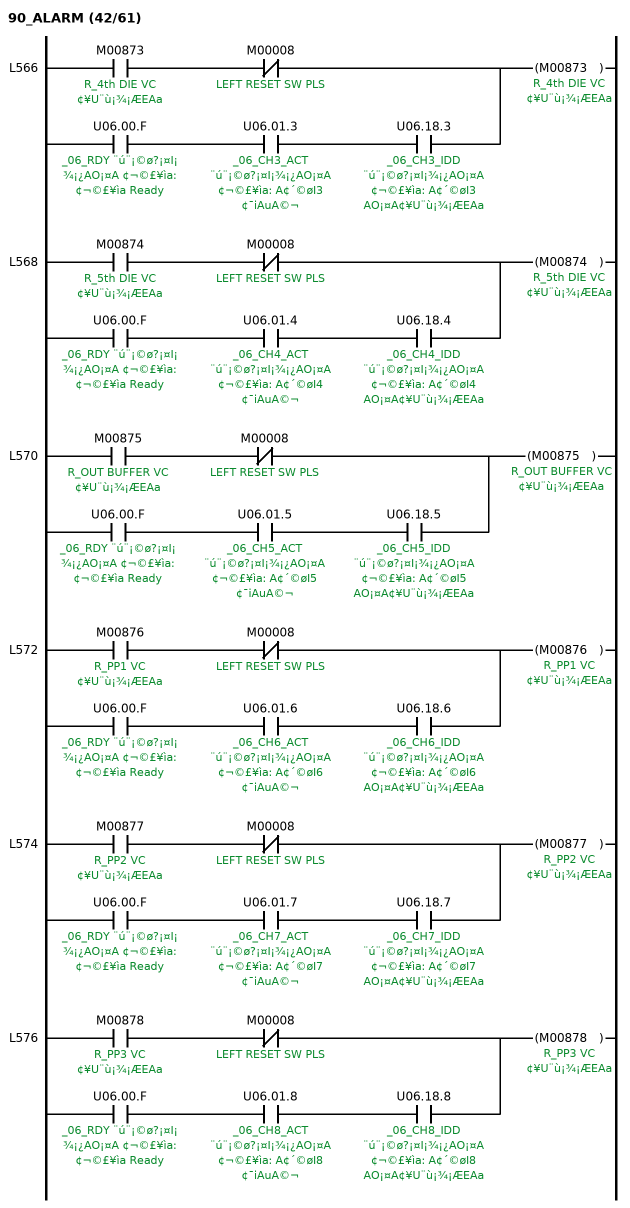
; L566
LOAD      M00873	// R_4th DIE VC ¢¥U¨ù¡¾¡ÆEAa
AND NOT   M00008	// LEFT RESET SW PLS
LOAD      U06.00.F	// _06_RDY ¨ú¨¡©ø?¡¤I¡¾¡¿AO¡¤A ¢¬©£¥ìa: ¢¬©£¥ìa Ready
AND       U06.01.3	// _06_CH3_ACT ¨ú¨¡©ø?¡¤I¡¾¡¿AO¡¤A ¢¬©£¥ìa: A¢´©øI3 ¢¯iAuA©¬
AND       U06.18.3	// _06_CH3_IDD ¨ú¨¡©ø?¡¤I¡¾¡¿AO¡¤A ¢¬©£¥ìa: A¢´©øI3 AO¡¤A¢¥U¨ù¡¾¡ÆEAa
OR LOAD
OUT       M00873	// R_4th DIE VC ¢¥U¨ù¡¾¡ÆEAa
; L568
LOAD      M00874	// R_5th DIE VC ¢¥U¨ù¡¾¡ÆEAa
AND NOT   M00008	// LEFT RESET SW PLS
LOAD      U06.00.F	// _06_RDY ¨ú¨¡©ø?¡¤I¡¾¡¿AO¡¤A ¢¬©£¥ìa: ¢¬©£¥ìa Ready
AND       U06.01.4	// _06_CH4_ACT ¨ú¨¡©ø?¡¤I¡¾¡¿AO¡¤A ¢¬©£¥ìa: A¢´©øI4 ¢¯iAuA©¬
AND       U06.18.4	// _06_CH4_IDD ¨ú¨¡©ø?¡¤I¡¾¡¿AO¡¤A ¢¬©£¥ìa: A¢´©øI4 AO¡¤A¢¥U¨ù¡¾¡ÆEAa
OR LOAD
OUT       M00874	// R_5th DIE VC ¢¥U¨ù¡¾¡ÆEAa
; L570
LOAD      M00875	// R_OUT BUFFER VC ¢¥U¨ù¡¾¡ÆEAa
AND NOT   M00008	// LEFT RESET SW PLS
LOAD      U06.00.F	// _06_RDY ¨ú¨¡©ø?¡¤I¡¾¡¿AO¡¤A ¢¬©£¥ìa: ¢¬©£¥ìa Ready
AND       U06.01.5	// _06_CH5_ACT ¨ú¨¡©ø?¡¤I¡¾¡¿AO¡¤A ¢¬©£¥ìa: A¢´©øI5 ¢¯iAuA©¬
AND       U06.18.5	// _06_CH5_IDD ¨ú¨¡©ø?¡¤I¡¾¡¿AO¡¤A ¢¬©£¥ìa: A¢´©øI5 AO¡¤A¢¥U¨ù¡¾¡ÆEAa
OR LOAD
OUT       M00875	// R_OUT BUFFER VC ¢¥U¨ù¡¾¡ÆEAa
; L572
LOAD      M00876	// R_PP1 VC ¢¥U¨ù¡¾¡ÆEAa
AND NOT   M00008	// LEFT RESET SW PLS
LOAD      U06.00.F	// _06_RDY ¨ú¨¡©ø?¡¤I¡¾¡¿AO¡¤A ¢¬©£¥ìa: ¢¬©£¥ìa Ready
AND       U06.01.6	// _06_CH6_ACT ¨ú¨¡©ø?¡¤I¡¾¡¿AO¡¤A ¢¬©£¥ìa: A¢´©øI6 ¢¯iAuA©¬
AND       U06.18.6	// _06_CH6_IDD ¨ú¨¡©ø?¡¤I¡¾¡¿AO¡¤A ¢¬©£¥ìa: A¢´©øI6 AO¡¤A¢¥U¨ù¡¾¡ÆEAa
OR LOAD
OUT       M00876	// R_PP1 VC ¢¥U¨ù¡¾¡ÆEAa
; L574
LOAD      M00877	// R_PP2 VC ¢¥U¨ù¡¾¡ÆEAa
AND NOT   M00008	// LEFT RESET SW PLS
LOAD      U06.00.F	// _06_RDY ¨ú¨¡©ø?¡¤I¡¾¡¿AO¡¤A ¢¬©£¥ìa: ¢¬©£¥ìa Ready
AND       U06.01.7	// _06_CH7_ACT ¨ú¨¡©ø?¡¤I¡¾¡¿AO¡¤A ¢¬©£¥ìa: A¢´©øI7 ¢¯iAuA©¬
AND       U06.18.7	// _06_CH7_IDD ¨ú¨¡©ø?¡¤I¡¾¡¿AO¡¤A ¢¬©£¥ìa: A¢´©øI7 AO¡¤A¢¥U¨ù¡¾¡ÆEAa
OR LOAD
OUT       M00877	// R_PP2 VC ¢¥U¨ù¡¾¡ÆEAa
; L576
LOAD      M00878	// R_PP3 VC ¢¥U¨ù¡¾¡ÆEAa
AND NOT   M00008	// LEFT RESET SW PLS
LOAD      U06.00.F	// _06_RDY ¨ú¨¡©ø?¡¤I¡¾¡¿AO¡¤A ¢¬©£¥ìa: ¢¬©£¥ìa Ready
AND       U06.01.8	// _06_CH8_ACT ¨ú¨¡©ø?¡¤I¡¾¡¿AO¡¤A ¢¬©£¥ìa: A¢´©øI8 ¢¯iAuA©¬
AND       U06.18.8	// _06_CH8_IDD ¨ú¨¡©ø?¡¤I¡¾¡¿AO¡¤A ¢¬©£¥ìa: A¢´©øI8 AO¡¤A¢¥U¨ù¡¾¡ÆEAa
OR LOAD
OUT       M00878	// R_PP3 VC ¢¥U¨ù¡¾¡ÆEAa

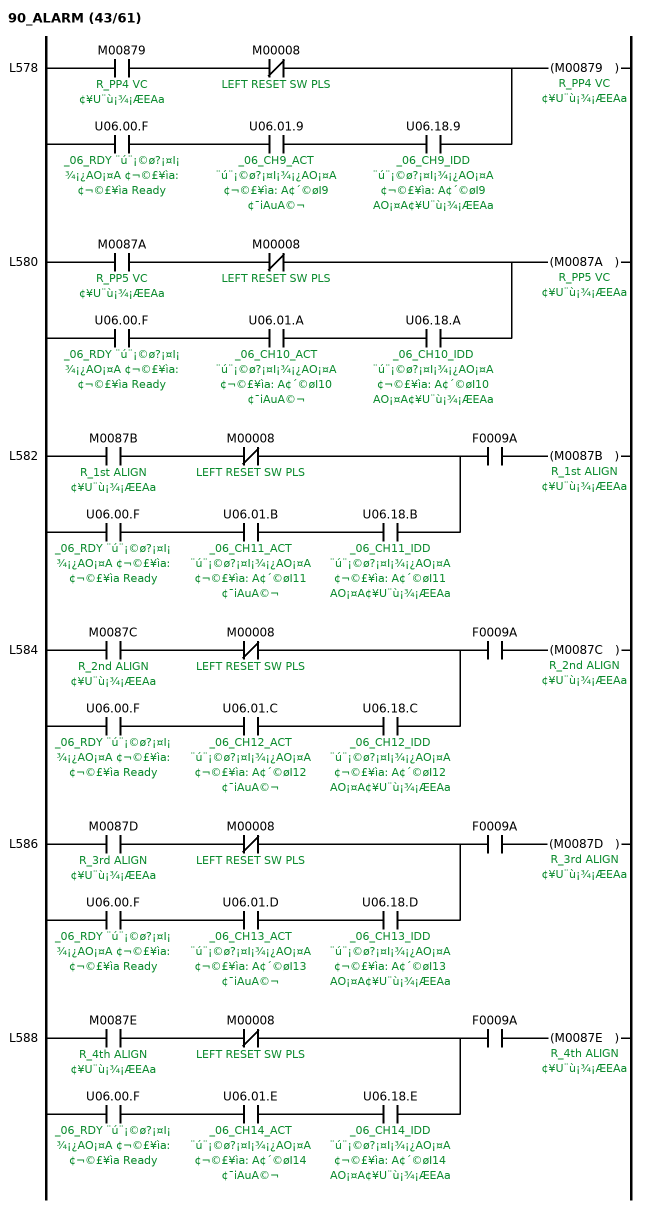
; L578
LOAD      M00879	// R_PP4 VC ¢¥U¨ù¡¾¡ÆEAa
AND NOT   M00008	// LEFT RESET SW PLS
LOAD      U06.00.F	// _06_RDY ¨ú¨¡©ø?¡¤I¡¾¡¿AO¡¤A ¢¬©£¥ìa: ¢¬©£¥ìa Ready
AND       U06.01.9	// _06_CH9_ACT ¨ú¨¡©ø?¡¤I¡¾¡¿AO¡¤A ¢¬©£¥ìa: A¢´©øI9 ¢¯iAuA©¬
AND       U06.18.9	// _06_CH9_IDD ¨ú¨¡©ø?¡¤I¡¾¡¿AO¡¤A ¢¬©£¥ìa: A¢´©øI9 AO¡¤A¢¥U¨ù¡¾¡ÆEAa
OR LOAD
OUT       M00879	// R_PP4 VC ¢¥U¨ù¡¾¡ÆEAa
; L580
LOAD      M0087A	// R_PP5 VC ¢¥U¨ù¡¾¡ÆEAa
AND NOT   M00008	// LEFT RESET SW PLS
LOAD      U06.00.F	// _06_RDY ¨ú¨¡©ø?¡¤I¡¾¡¿AO¡¤A ¢¬©£¥ìa: ¢¬©£¥ìa Ready
AND       U06.01.A	// _06_CH10_ACT ¨ú¨¡©ø?¡¤I¡¾¡¿AO¡¤A ¢¬©£¥ìa: A¢´©øI10 ¢¯iAuA©¬
AND       U06.18.A	// _06_CH10_IDD ¨ú¨¡©ø?¡¤I¡¾¡¿AO¡¤A ¢¬©£¥ìa: A¢´©øI10 AO¡¤A¢¥U¨ù¡¾¡ÆEAa
OR LOAD
OUT       M0087A	// R_PP5 VC ¢¥U¨ù¡¾¡ÆEAa
; L582
LOAD      M0087B	// R_1st ALIGN ¢¥U¨ù¡¾¡ÆEAa
AND NOT   M00008	// LEFT RESET SW PLS
LOAD      U06.00.F	// _06_RDY ¨ú¨¡©ø?¡¤I¡¾¡¿AO¡¤A ¢¬©£¥ìa: ¢¬©£¥ìa Ready
AND       U06.01.B	// _06_CH11_ACT ¨ú¨¡©ø?¡¤I¡¾¡¿AO¡¤A ¢¬©£¥ìa: A¢´©øI11 ¢¯iAuA©¬
AND       U06.18.B	// _06_CH11_IDD ¨ú¨¡©ø?¡¤I¡¾¡¿AO¡¤A ¢¬©£¥ìa: A¢´©øI11 AO¡¤A¢¥U¨ù¡¾¡ÆEAa
OR LOAD
AND       F0009A
OUT       M0087B	// R_1st ALIGN ¢¥U¨ù¡¾¡ÆEAa
; L584
LOAD      M0087C	// R_2nd ALIGN ¢¥U¨ù¡¾¡ÆEAa
AND NOT   M00008	// LEFT RESET SW PLS
LOAD      U06.00.F	// _06_RDY ¨ú¨¡©ø?¡¤I¡¾¡¿AO¡¤A ¢¬©£¥ìa: ¢¬©£¥ìa Ready
AND       U06.01.C	// _06_CH12_ACT ¨ú¨¡©ø?¡¤I¡¾¡¿AO¡¤A ¢¬©£¥ìa: A¢´©øI12 ¢¯iAuA©¬
AND       U06.18.C	// _06_CH12_IDD ¨ú¨¡©ø?¡¤I¡¾¡¿AO¡¤A ¢¬©£¥ìa: A¢´©øI12 AO¡¤A¢¥U¨ù¡¾¡ÆEAa
OR LOAD
AND       F0009A
OUT       M0087C	// R_2nd ALIGN ¢¥U¨ù¡¾¡ÆEAa
; L586
LOAD      M0087D	// R_3rd ALIGN ¢¥U¨ù¡¾¡ÆEAa
AND NOT   M00008	// LEFT RESET SW PLS
LOAD      U06.00.F	// _06_RDY ¨ú¨¡©ø?¡¤I¡¾¡¿AO¡¤A ¢¬©£¥ìa: ¢¬©£¥ìa Ready
AND       U06.01.D	// _06_CH13_ACT ¨ú¨¡©ø?¡¤I¡¾¡¿AO¡¤A ¢¬©£¥ìa: A¢´©øI13 ¢¯iAuA©¬
AND       U06.18.D	// _06_CH13_IDD ¨ú¨¡©ø?¡¤I¡¾¡¿AO¡¤A ¢¬©£¥ìa: A¢´©øI13 AO¡¤A¢¥U¨ù¡¾¡ÆEAa
OR LOAD
AND       F0009A
OUT       M0087D	// R_3rd ALIGN ¢¥U¨ù¡¾¡ÆEAa
; L588
LOAD      M0087E	// R_4th ALIGN ¢¥U¨ù¡¾¡ÆEAa
AND NOT   M00008	// LEFT RESET SW PLS
LOAD      U06.00.F	// _06_RDY ¨ú¨¡©ø?¡¤I¡¾¡¿AO¡¤A ¢¬©£¥ìa: ¢¬©£¥ìa Ready
AND       U06.01.E	// _06_CH14_ACT ¨ú¨¡©ø?¡¤I¡¾¡¿AO¡¤A ¢¬©£¥ìa: A¢´©øI14 ¢¯iAuA©¬
AND       U06.18.E	// _06_CH14_IDD ¨ú¨¡©ø?¡¤I¡¾¡¿AO¡¤A ¢¬©£¥ìa: A¢´©øI14 AO¡¤A¢¥U¨ù¡¾¡ÆEAa
OR LOAD
AND       F0009A
OUT       M0087E	// R_4th ALIGN ¢¥U¨ù¡¾¡ÆEAa

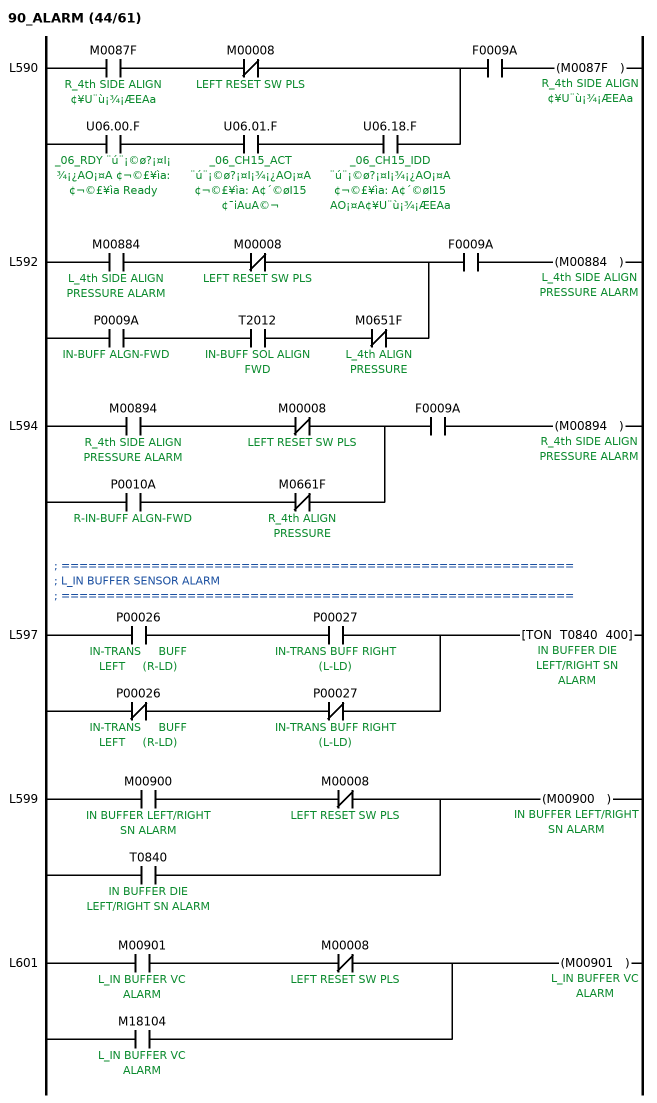
; L590
LOAD      M0087F	// R_4th SIDE ALIGN ¢¥U¨ù¡¾¡ÆEAa
AND NOT   M00008	// LEFT RESET SW PLS
LOAD      U06.00.F	// _06_RDY ¨ú¨¡©ø?¡¤I¡¾¡¿AO¡¤A ¢¬©£¥ìa: ¢¬©£¥ìa Ready
AND       U06.01.F	// _06_CH15_ACT ¨ú¨¡©ø?¡¤I¡¾¡¿AO¡¤A ¢¬©£¥ìa: A¢´©øI15 ¢¯iAuA©¬
AND       U06.18.F	// _06_CH15_IDD ¨ú¨¡©ø?¡¤I¡¾¡¿AO¡¤A ¢¬©£¥ìa: A¢´©øI15 AO¡¤A¢¥U¨ù¡¾¡ÆEAa
OR LOAD
AND       F0009A
OUT       M0087F	// R_4th SIDE ALIGN ¢¥U¨ù¡¾¡ÆEAa
; L592
LOAD      M00884	// L_4th SIDE ALIGN PRESSURE ALARM
AND NOT   M00008	// LEFT RESET SW PLS
LOAD      P0009A	// IN-BUFF ALGN-FWD
AND       T2012	// IN-BUFF SOL ALIGN FWD
AND NOT   M0651F	// L_4th ALIGN PRESSURE
OR LOAD
AND       F0009A
OUT       M00884	// L_4th SIDE ALIGN PRESSURE ALARM
; L594
LOAD      M00894	// R_4th SIDE ALIGN PRESSURE ALARM
AND NOT   M00008	// LEFT RESET SW PLS
LOAD      P0010A	// R-IN-BUFF ALGN-FWD
AND NOT   M0661F	// R_4th ALIGN PRESSURE
OR LOAD
AND       F0009A
OUT       M00894	// R_4th SIDE ALIGN PRESSURE ALARM
// =========================================================
// 
//        L_IN BUFFER SENSOR ALARM
// 
// =========================================================
; L597
LOAD      P00026	// IN-TRANS     BUFF     LEFT     (R-LD)
AND       P00027	// IN-TRANS BUFF RIGHT     (L-LD)
LOAD NOT  P00026	// IN-TRANS     BUFF     LEFT     (R-LD)
AND NOT   P00027	// IN-TRANS BUFF RIGHT     (L-LD)
OR LOAD
TON       T0840 400	// IN BUFFER DIE LEFT/RIGHT SN ALARM
; L599
LOAD      M00900	// IN BUFFER LEFT/RIGHT SN ALARM
AND NOT   M00008	// LEFT RESET SW PLS
OR        T0840	// IN BUFFER DIE LEFT/RIGHT SN ALARM
OUT       M00900	// IN BUFFER LEFT/RIGHT SN ALARM
; L601
LOAD      M00901	// L_IN BUFFER VC ALARM
AND NOT   M00008	// LEFT RESET SW PLS
OR        M18104	// L_IN BUFFER VC ALARM
OUT       M00901	// L_IN BUFFER VC ALARM

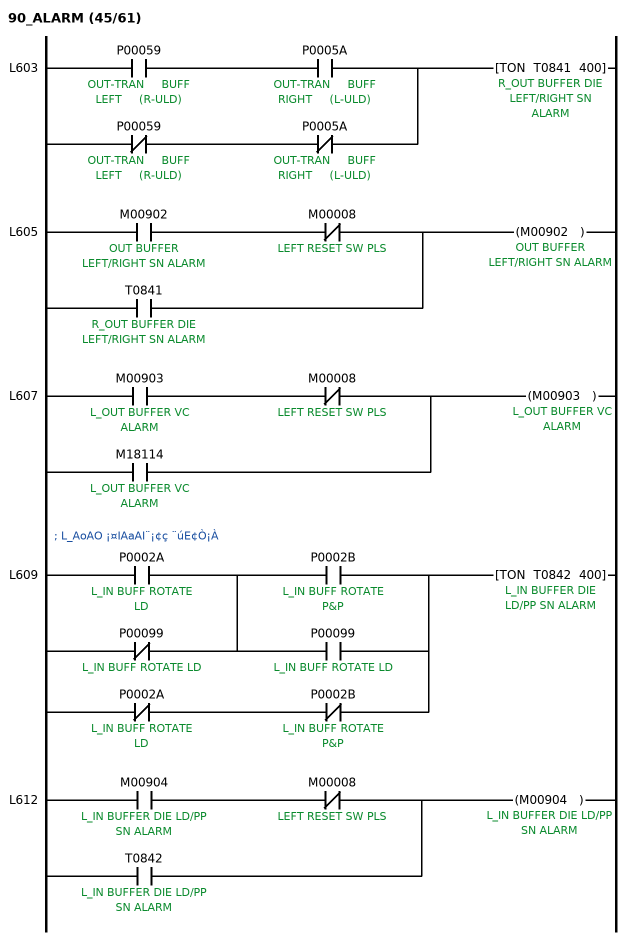
; L603
LOAD      P00059	// OUT-TRAN     BUFF     LEFT     (R-ULD)
AND       P0005A	// OUT-TRAN     BUFF     RIGHT     (L-ULD)
LOAD NOT  P00059	// OUT-TRAN     BUFF     LEFT     (R-ULD)
AND NOT   P0005A	// OUT-TRAN     BUFF     RIGHT     (L-ULD)
OR LOAD
TON       T0841 400	// R_OUT BUFFER DIE LEFT/RIGHT SN ALARM
; L605
LOAD      M00902	// OUT BUFFER LEFT/RIGHT SN ALARM
AND NOT   M00008	// LEFT RESET SW PLS
OR        T0841	// R_OUT BUFFER DIE LEFT/RIGHT SN ALARM
OUT       M00902	// OUT BUFFER LEFT/RIGHT SN ALARM
; L607
LOAD      M00903	// L_OUT BUFFER VC ALARM
AND NOT   M00008	// LEFT RESET SW PLS
OR        M18114	// L_OUT BUFFER VC ALARM
OUT       M00903	// L_OUT BUFFER VC ALARM
; L609
LOAD      P0002A	// L_IN BUFF ROTATE     LD
OR NOT    P00099	// L_IN BUFF ROTATE LD
LOAD      P0002B	// L_IN BUFF ROTATE      P&P
OR        P00099	// L_IN BUFF ROTATE LD
AND LOAD
LOAD NOT  P0002A	// L_IN BUFF ROTATE     LD
AND NOT   P0002B	// L_IN BUFF ROTATE      P&P
OR LOAD
TON       T0842 400	// L_IN BUFFER DIE LD/PP SN ALARM
// output comment: L_AoAO ¡¤IAaAI¨¡¢ç ¨úE¢Ò¡À
; L612
LOAD      M00904	// L_IN BUFFER DIE LD/PP SN ALARM
AND NOT   M00008	// LEFT RESET SW PLS
OR        T0842	// L_IN BUFFER DIE LD/PP SN ALARM
OUT       M00904	// L_IN BUFFER DIE LD/PP SN ALARM

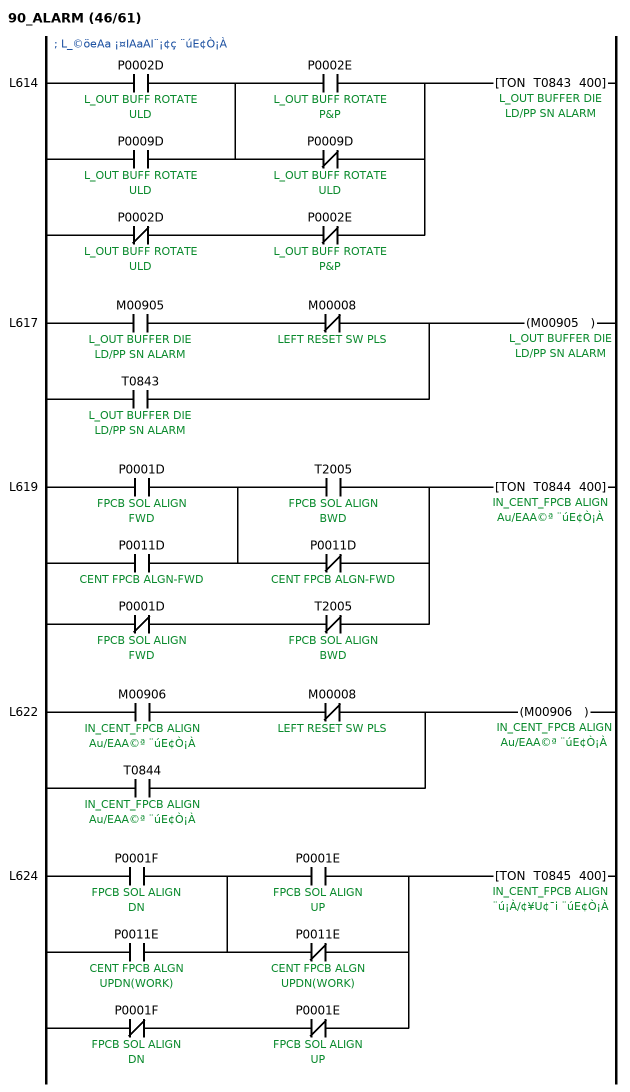
; L614
LOAD      P0002D	// L_OUT BUFF ROTATE     ULD
OR        P0009D	// L_OUT BUFF ROTATE ULD
LOAD      P0002E	// L_OUT BUFF ROTATE      P&P
OR NOT    P0009D	// L_OUT BUFF ROTATE ULD
AND LOAD
LOAD NOT  P0002D	// L_OUT BUFF ROTATE     ULD
AND NOT   P0002E	// L_OUT BUFF ROTATE      P&P
OR LOAD
TON       T0843 400	// L_OUT BUFFER DIE LD/PP SN ALARM
// output comment: L_©öeAa ¡¤IAaAI¨¡¢ç ¨úE¢Ò¡À
; L617
LOAD      M00905	// L_OUT BUFFER DIE LD/PP SN ALARM
AND NOT   M00008	// LEFT RESET SW PLS
OR        T0843	// L_OUT BUFFER DIE LD/PP SN ALARM
OUT       M00905	// L_OUT BUFFER DIE LD/PP SN ALARM
; L619
LOAD      P0001D	// FPCB SOL ALIGN         FWD
OR        P0011D	// CENT FPCB ALGN-FWD
LOAD      T2005	// FPCB SOL ALIGN         BWD
OR NOT    P0011D	// CENT FPCB ALGN-FWD
AND LOAD
LOAD NOT  P0001D	// FPCB SOL ALIGN         FWD
AND NOT   T2005	// FPCB SOL ALIGN         BWD
OR LOAD
TON       T0844 400	// IN_CENT_FPCB ALIGN Au/EAA©ª ¨úE¢Ò¡À
; L622
LOAD      M00906	// IN_CENT_FPCB ALIGN Au/EAA©ª ¨úE¢Ò¡À
AND NOT   M00008	// LEFT RESET SW PLS
OR        T0844	// IN_CENT_FPCB ALIGN Au/EAA©ª ¨úE¢Ò¡À
OUT       M00906	// IN_CENT_FPCB ALIGN Au/EAA©ª ¨úE¢Ò¡À
; L624
LOAD      P0001F	// FPCB SOL ALIGN        DN
OR        P0011E	// CENT FPCB ALGN UPDN(WORK)
LOAD      P0001E	// FPCB SOL ALIGN         UP
OR NOT    P0011E	// CENT FPCB ALGN UPDN(WORK)
AND LOAD
LOAD NOT  P0001F	// FPCB SOL ALIGN        DN
AND NOT   P0001E	// FPCB SOL ALIGN         UP
OR LOAD
TON       T0845 400	// IN_CENT_FPCB ALIGN ¨ú¡À/¢¥U¢¯i ¨úE¢Ò¡À

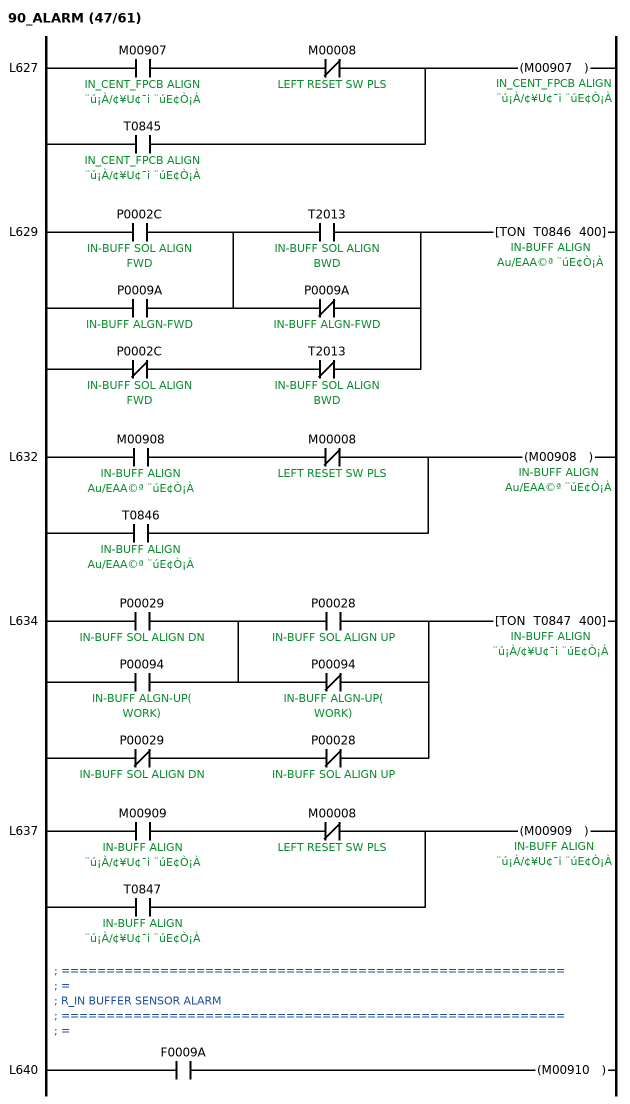
; L627
LOAD      M00907	// IN_CENT_FPCB ALIGN ¨ú¡À/¢¥U¢¯i ¨úE¢Ò¡À
AND NOT   M00008	// LEFT RESET SW PLS
OR        T0845	// IN_CENT_FPCB ALIGN ¨ú¡À/¢¥U¢¯i ¨úE¢Ò¡À
OUT       M00907	// IN_CENT_FPCB ALIGN ¨ú¡À/¢¥U¢¯i ¨úE¢Ò¡À
; L629
LOAD      P0002C	// IN-BUFF SOL ALIGN FWD
OR        P0009A	// IN-BUFF ALGN-FWD
LOAD      T2013	// IN-BUFF SOL ALIGN BWD
OR NOT    P0009A	// IN-BUFF ALGN-FWD
AND LOAD
LOAD NOT  P0002C	// IN-BUFF SOL ALIGN FWD
AND NOT   T2013	// IN-BUFF SOL ALIGN BWD
OR LOAD
TON       T0846 400	// IN-BUFF ALIGN Au/EAA©ª ¨úE¢Ò¡À
; L632
LOAD      M00908	// IN-BUFF ALIGN Au/EAA©ª ¨úE¢Ò¡À
AND NOT   M00008	// LEFT RESET SW PLS
OR        T0846	// IN-BUFF ALIGN Au/EAA©ª ¨úE¢Ò¡À
OUT       M00908	// IN-BUFF ALIGN Au/EAA©ª ¨úE¢Ò¡À
; L634
LOAD      P00029	// IN-BUFF SOL ALIGN DN
OR        P00094	// IN-BUFF ALGN-UP(WORK)
LOAD      P00028	// IN-BUFF SOL ALIGN UP
OR NOT    P00094	// IN-BUFF ALGN-UP(WORK)
AND LOAD
LOAD NOT  P00029	// IN-BUFF SOL ALIGN DN
AND NOT   P00028	// IN-BUFF SOL ALIGN UP
OR LOAD
TON       T0847 400	// IN-BUFF ALIGN ¨ú¡À/¢¥U¢¯i ¨úE¢Ò¡À
; L637
LOAD      M00909	// IN-BUFF ALIGN ¨ú¡À/¢¥U¢¯i ¨úE¢Ò¡À
AND NOT   M00008	// LEFT RESET SW PLS
OR        T0847	// IN-BUFF ALIGN ¨ú¡À/¢¥U¢¯i ¨úE¢Ò¡À
OUT       M00909	// IN-BUFF ALIGN ¨ú¡À/¢¥U¢¯i ¨úE¢Ò¡À
// =========================================================
// 
//        R_IN BUFFER SENSOR ALARM
// 
// =========================================================
; L640
LOAD      F0009A
OUT       M00910

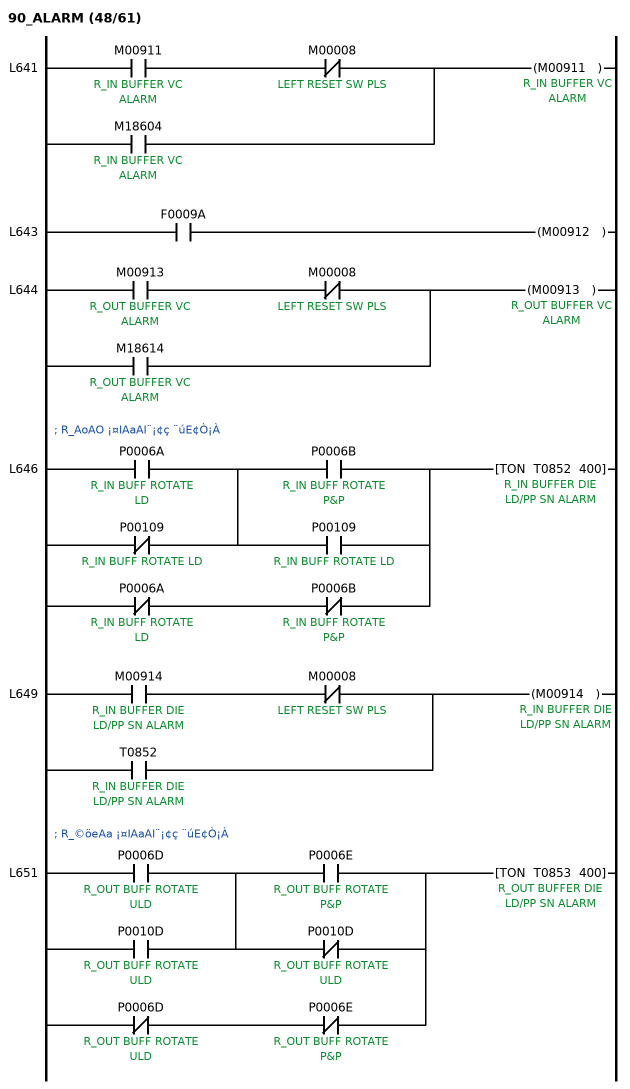
; L641
LOAD      M00911	// R_IN BUFFER VC ALARM
AND NOT   M00008	// LEFT RESET SW PLS
OR        M18604	// R_IN BUFFER VC ALARM
OUT       M00911	// R_IN BUFFER VC ALARM
; L643
LOAD      F0009A
OUT       M00912
; L644
LOAD      M00913	// R_OUT BUFFER VC ALARM
AND NOT   M00008	// LEFT RESET SW PLS
OR        M18614	// R_OUT BUFFER VC ALARM
OUT       M00913	// R_OUT BUFFER VC ALARM
; L646
LOAD      P0006A	// R_IN BUFF ROTATE      LD
OR NOT    P00109	// R_IN BUFF ROTATE LD
LOAD      P0006B	// R_IN BUFF ROTATE      P&P
OR        P00109	// R_IN BUFF ROTATE LD
AND LOAD
LOAD NOT  P0006A	// R_IN BUFF ROTATE      LD
AND NOT   P0006B	// R_IN BUFF ROTATE      P&P
OR LOAD
TON       T0852 400	// R_IN BUFFER DIE LD/PP SN ALARM
// output comment: R_AoAO ¡¤IAaAI¨¡¢ç ¨úE¢Ò¡À
; L649
LOAD      M00914	// R_IN BUFFER DIE LD/PP SN ALARM
AND NOT   M00008	// LEFT RESET SW PLS
OR        T0852	// R_IN BUFFER DIE LD/PP SN ALARM
OUT       M00914	// R_IN BUFFER DIE LD/PP SN ALARM
; L651
LOAD      P0006D	// R_OUT BUFF ROTATE      ULD
OR        P0010D	// R_OUT BUFF ROTATE ULD
LOAD      P0006E	// R_OUT BUFF ROTATE      P&P
OR NOT    P0010D	// R_OUT BUFF ROTATE ULD
AND LOAD
LOAD NOT  P0006D	// R_OUT BUFF ROTATE      ULD
AND NOT   P0006E	// R_OUT BUFF ROTATE      P&P
OR LOAD
TON       T0853 400	// R_OUT BUFFER DIE LD/PP SN ALARM
// output comment: R_©öeAa ¡¤IAaAI¨¡¢ç ¨úE¢Ò¡À

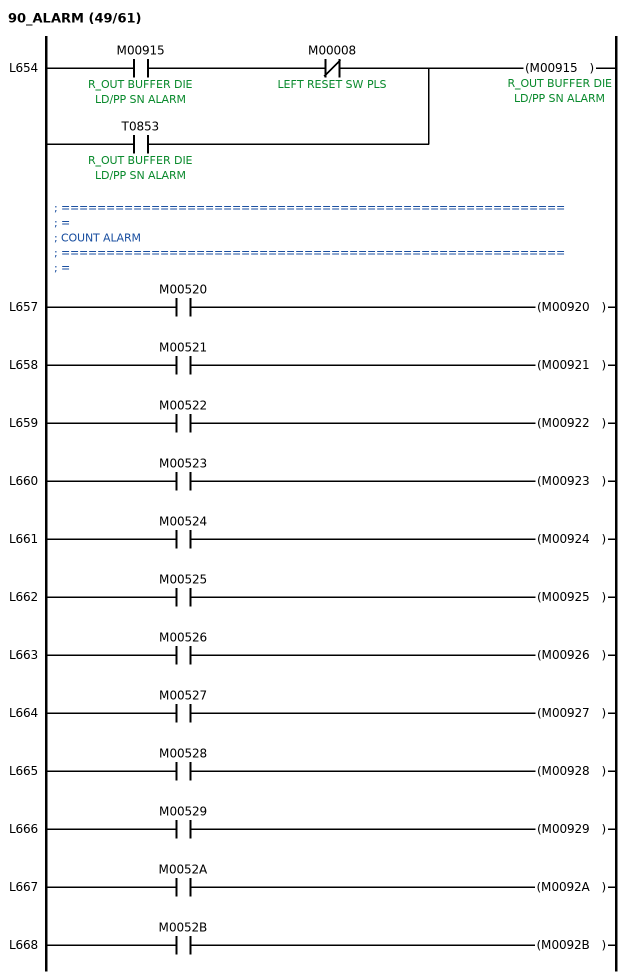
; L654
LOAD      M00915	// R_OUT BUFFER DIE LD/PP SN ALARM
AND NOT   M00008	// LEFT RESET SW PLS
OR        T0853	// R_OUT BUFFER DIE LD/PP SN ALARM
OUT       M00915	// R_OUT BUFFER DIE LD/PP SN ALARM
// =========================================================
// 
//       COUNT ALARM
// 
// =========================================================
; L657
LOAD      M00520
OUT       M00920
; L658
LOAD      M00521
OUT       M00921
; L659
LOAD      M00522
OUT       M00922
; L660
LOAD      M00523
OUT       M00923
; L661
LOAD      M00524
OUT       M00924
; L662
LOAD      M00525
OUT       M00925
; L663
LOAD      M00526
OUT       M00926
; L664
LOAD      M00527
OUT       M00927
; L665
LOAD      M00528
OUT       M00928
; L666
LOAD      M00529
OUT       M00929
; L667
LOAD      M0052A
OUT       M0092A
; L668
LOAD      M0052B
OUT       M0092B

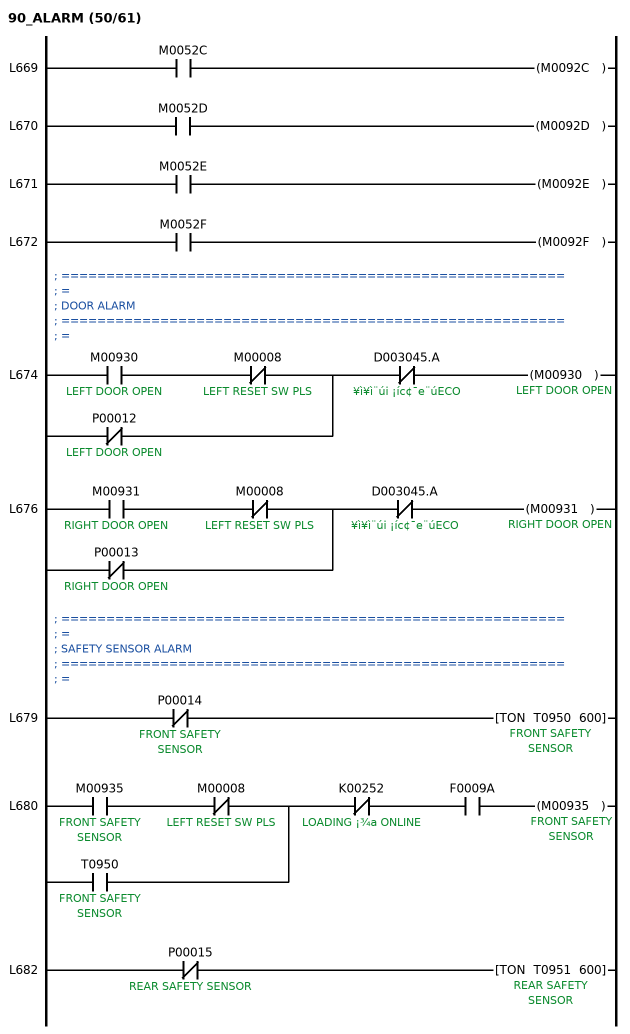
; L669
LOAD      M0052C
OUT       M0092C
; L670
LOAD      M0052D
OUT       M0092D
; L671
LOAD      M0052E
OUT       M0092E
; L672
LOAD      M0052F
OUT       M0092F
// =========================================================
// 
//       DOOR ALARM
// 
// =========================================================
; L674
LOAD      M00930	// LEFT DOOR OPEN
AND NOT   M00008	// LEFT RESET SW PLS
OR NOT    P00012	// LEFT DOOR OPEN
AND NOT   D003045.A	// ¥ì¥ì¨úi ¡íc¢¯e¨úECO
OUT       M00930	// LEFT DOOR OPEN
; L676
LOAD      M00931	// RIGHT DOOR OPEN
AND NOT   M00008	// LEFT RESET SW PLS
OR NOT    P00013	// RIGHT DOOR OPEN
AND NOT   D003045.A	// ¥ì¥ì¨úi ¡íc¢¯e¨úECO
OUT       M00931	// RIGHT DOOR OPEN
// =========================================================
// 
//       SAFETY SENSOR ALARM
// 
// =========================================================
; L679
LOAD NOT  P00014	// FRONT SAFETY SENSOR
TON       T0950 600	// FRONT SAFETY SENSOR
; L680
LOAD      M00935	// FRONT SAFETY SENSOR
AND NOT   M00008	// LEFT RESET SW PLS
OR        T0950	// FRONT SAFETY SENSOR
AND NOT   K00252	// LOADING ¡¾a ONLINE
AND       F0009A
OUT       M00935	// FRONT SAFETY SENSOR
; L682
LOAD NOT  P00015	// REAR SAFETY SENSOR
TON       T0951 600	// REAR SAFETY SENSOR

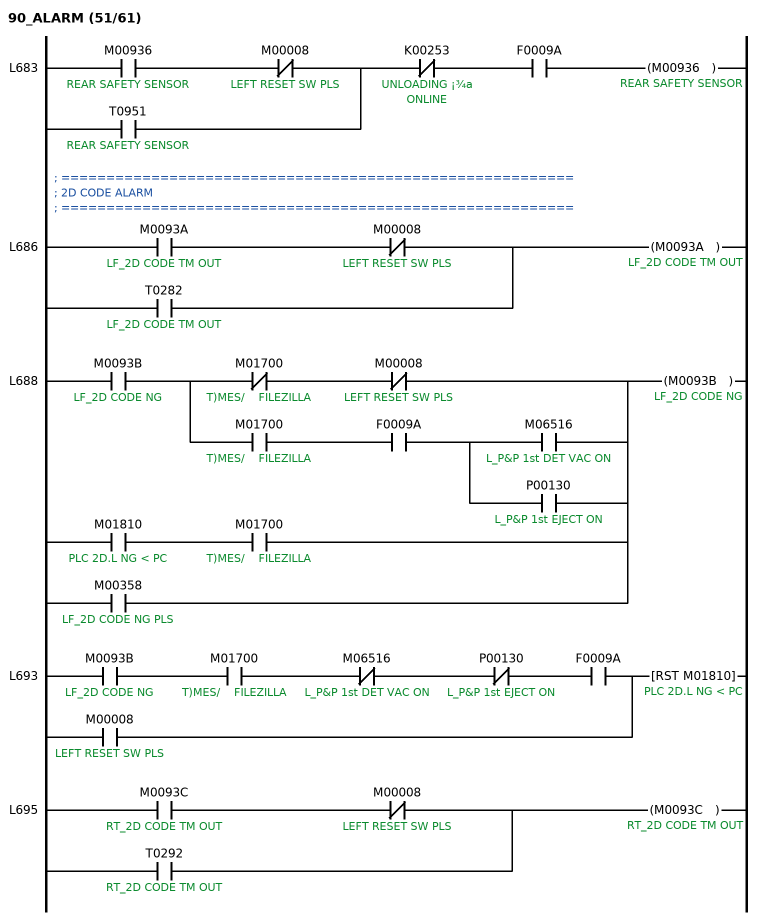
; L683
LOAD      M00936	// REAR SAFETY SENSOR
AND NOT   M00008	// LEFT RESET SW PLS
OR        T0951	// REAR SAFETY SENSOR
AND NOT   K00253	// UNLOADING ¡¾a ONLINE
AND       F0009A
OUT       M00936	// REAR SAFETY SENSOR
// =========================================================
// 
//       2D CODE ALARM
// 
// =========================================================
; L686
LOAD      M0093A	// LF_2D CODE TM OUT
AND NOT   M00008	// LEFT RESET SW PLS
OR        T0282	// LF_2D CODE TM OUT
OUT       M0093A	// LF_2D CODE TM OUT
; L688
LOAD      M0093B	// LF_2D CODE NG
LOAD NOT  M01700	// T)MES/    FILEZILLA
AND NOT   M00008	// LEFT RESET SW PLS
LOAD      M01700	// T)MES/    FILEZILLA
AND       F0009A
LOAD      M06516	// L_P&P 1st DET VAC ON
OR        P00130	// L_P&P 1st EJECT ON
AND LOAD
OR LOAD
AND LOAD
LOAD      M01810	// PLC 2D.L NG < PC
AND       M01700	// T)MES/    FILEZILLA
OR LOAD
OR        M00358	// LF_2D CODE NG PLS
OUT       M0093B	// LF_2D CODE NG
; L693
LOAD      M0093B	// LF_2D CODE NG
AND       M01700	// T)MES/    FILEZILLA
AND NOT   M06516	// L_P&P 1st DET VAC ON
AND NOT   P00130	// L_P&P 1st EJECT ON
AND       F0009A
OR        M00008	// LEFT RESET SW PLS
RST       M01810	// PLC 2D.L NG < PC
; L695
LOAD      M0093C	// RT_2D CODE TM OUT
AND NOT   M00008	// LEFT RESET SW PLS
OR        T0292	// RT_2D CODE TM OUT
OUT       M0093C	// RT_2D CODE TM OUT

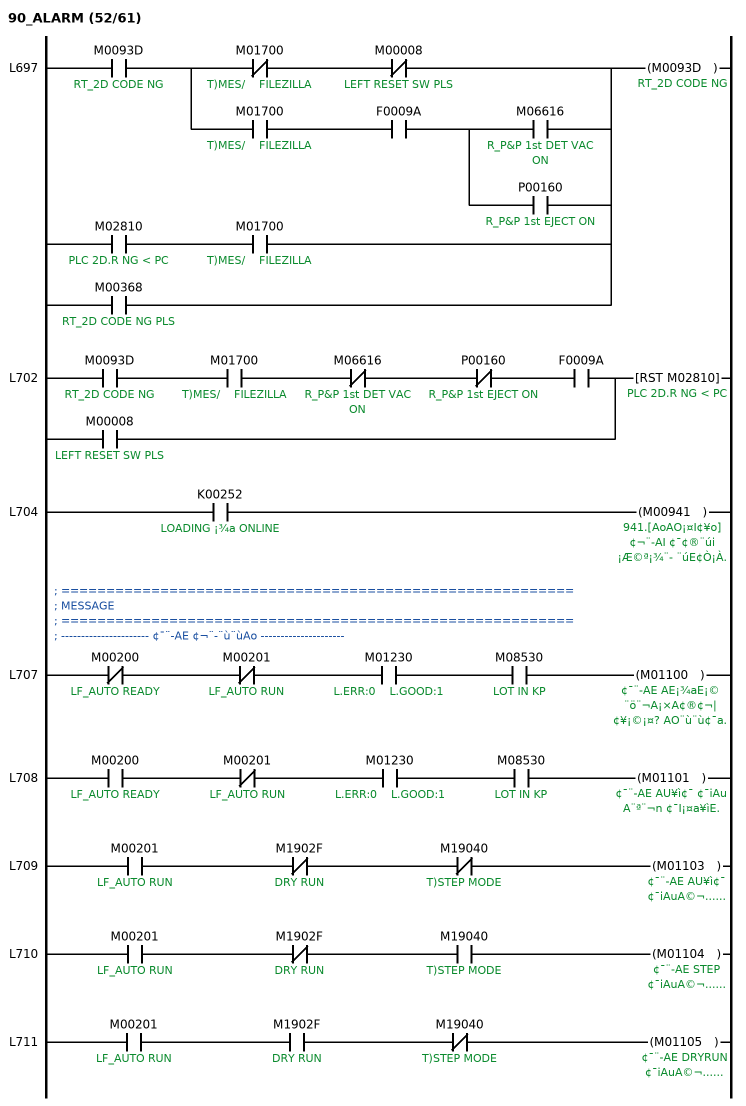
; L697
LOAD      M0093D	// RT_2D CODE NG
LOAD NOT  M01700	// T)MES/    FILEZILLA
AND NOT   M00008	// LEFT RESET SW PLS
LOAD      M01700	// T)MES/    FILEZILLA
AND       F0009A
LOAD      M06616	// R_P&P 1st DET VAC ON
OR        P00160	// R_P&P 1st EJECT ON
AND LOAD
OR LOAD
AND LOAD
LOAD      M02810	// PLC 2D.R NG < PC
AND       M01700	// T)MES/    FILEZILLA
OR LOAD
OR        M00368	// RT_2D CODE NG PLS
OUT       M0093D	// RT_2D CODE NG
; L702
LOAD      M0093D	// RT_2D CODE NG
AND       M01700	// T)MES/    FILEZILLA
AND NOT   M06616	// R_P&P 1st DET VAC ON
AND NOT   P00160	// R_P&P 1st EJECT ON
AND       F0009A
OR        M00008	// LEFT RESET SW PLS
RST       M02810	// PLC 2D.R NG < PC
; L704
LOAD      K00252	// LOADING ¡¾a ONLINE
OUT       M00941	// 941.[AoAO¡¤I¢¥o] ¢¬¨­AI ¢¯¢®¨úi ¡Æ©ª¡¾¨­ ¨úE¢Ò¡À.
// =========================================================
// 
//       MESSAGE
// 
// =========================================================
// ---------------------- ¢¯¨­AE ¢¬¨­¨ù¨ùAo ---------------------
; L707
LOAD NOT  M00200	// LF_AUTO READY
AND NOT   M00201	// LF_AUTO RUN
AND       M01230	// L.ERR:0    L.GOOD:1
AND       M08530	// LOT IN KP
OUT       M01100	// ¢¯¨­AE AE¡¾aE¡© ¨ö¨¬A¡×A¢®¢¬| ¢¥¡©¡¤? AO¨ù¨ù¢¯a.
; L708
LOAD      M00200	// LF_AUTO READY
AND NOT   M00201	// LF_AUTO RUN
AND       M01230	// L.ERR:0    L.GOOD:1
AND       M08530	// LOT IN KP
OUT       M01101	// ¢¯¨­AE AU¥ì¢¯ ¢¯iAu A¨ª¨¬n ¢¯I¡¤a¥ìE.
; L709
LOAD      M00201	// LF_AUTO RUN
AND NOT   M1902F	// DRY RUN
AND NOT   M19040	// T)STEP MODE
OUT       M01103	// ¢¯¨­AE AU¥ì¢¯ ¢¯iAuA©¬......
; L710
LOAD      M00201	// LF_AUTO RUN
AND NOT   M1902F	// DRY RUN
AND       M19040	// T)STEP MODE
OUT       M01104	// ¢¯¨­AE STEP ¢¯iAuA©¬......
; L711
LOAD      M00201	// LF_AUTO RUN
AND       M1902F	// DRY RUN
AND NOT   M19040	// T)STEP MODE
OUT       M01105	// ¢¯¨­AE DRYRUN ¢¯iAuA©¬......

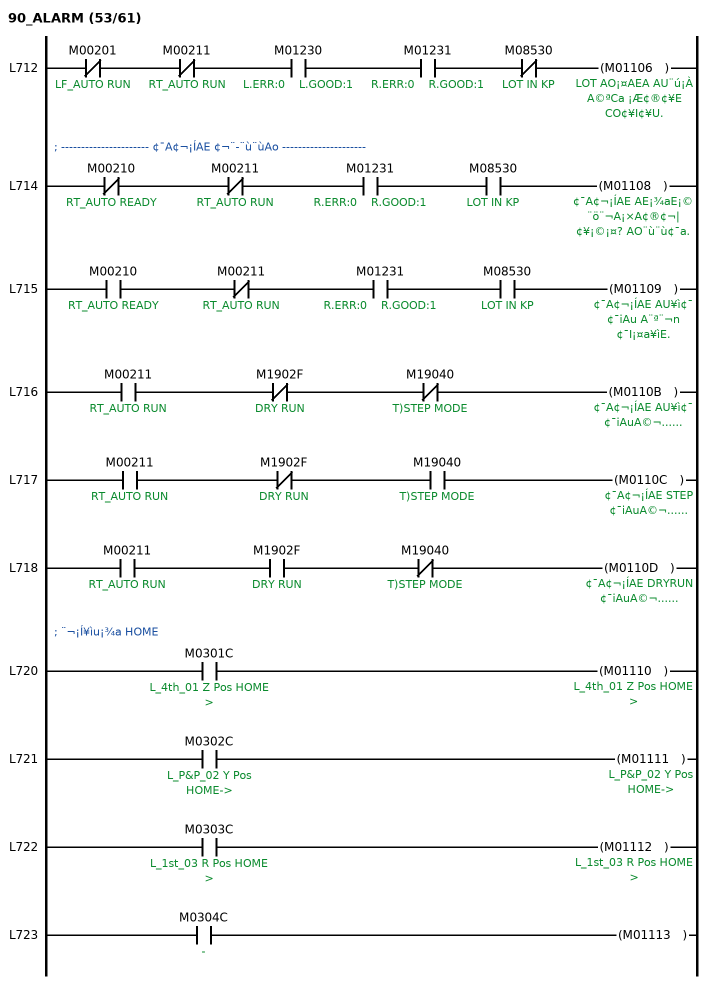
; L712
LOAD NOT  M00201	// LF_AUTO RUN
AND NOT   M00211	// RT_AUTO RUN
AND       M01230	// L.ERR:0    L.GOOD:1
AND       M01231	// R.ERR:0    R.GOOD:1
AND NOT   M08530	// LOT IN KP
OUT       M01106	// LOT AO¡¤AEA AU¨ú¡À A©ªCa ¡Æ¢®¢¥E CO¢¥I¢¥U.
// ---------------------- ¢¯A¢¬¡ÍAE ¢¬¨­¨ù¨ùAo ---------------------
; L714
LOAD NOT  M00210	// RT_AUTO READY
AND NOT   M00211	// RT_AUTO RUN
AND       M01231	// R.ERR:0    R.GOOD:1
AND       M08530	// LOT IN KP
OUT       M01108	// ¢¯A¢¬¡ÍAE AE¡¾aE¡© ¨ö¨¬A¡×A¢®¢¬| ¢¥¡©¡¤? AO¨ù¨ù¢¯a.
; L715
LOAD      M00210	// RT_AUTO READY
AND NOT   M00211	// RT_AUTO RUN
AND       M01231	// R.ERR:0    R.GOOD:1
AND       M08530	// LOT IN KP
OUT       M01109	// ¢¯A¢¬¡ÍAE AU¥ì¢¯ ¢¯iAu A¨ª¨¬n ¢¯I¡¤a¥ìE.
; L716
LOAD      M00211	// RT_AUTO RUN
AND NOT   M1902F	// DRY RUN
AND NOT   M19040	// T)STEP MODE
OUT       M0110B	// ¢¯A¢¬¡ÍAE AU¥ì¢¯ ¢¯iAuA©¬......
; L717
LOAD      M00211	// RT_AUTO RUN
AND NOT   M1902F	// DRY RUN
AND       M19040	// T)STEP MODE
OUT       M0110C	// ¢¯A¢¬¡ÍAE STEP ¢¯iAuA©¬......
; L718
LOAD      M00211	// RT_AUTO RUN
AND       M1902F	// DRY RUN
AND NOT   M19040	// T)STEP MODE
OUT       M0110D	// ¢¯A¢¬¡ÍAE DRYRUN ¢¯iAuA©¬......
// ¨¬¡Í¥ìu¡¾a HOME
; L720
LOAD      M0301C	// L_4th_01 Z Pos HOME >
OUT       M01110	// L_4th_01 Z Pos HOME >
; L721
LOAD      M0302C	// L_P&P_02 Y Pos HOME->
OUT       M01111	// L_P&P_02 Y Pos HOME->
; L722
LOAD      M0303C	// L_1st_03 R Pos HOME >
OUT       M01112	// L_1st_03 R Pos HOME >
; L723
LOAD      M0304C	// -
OUT       M01113

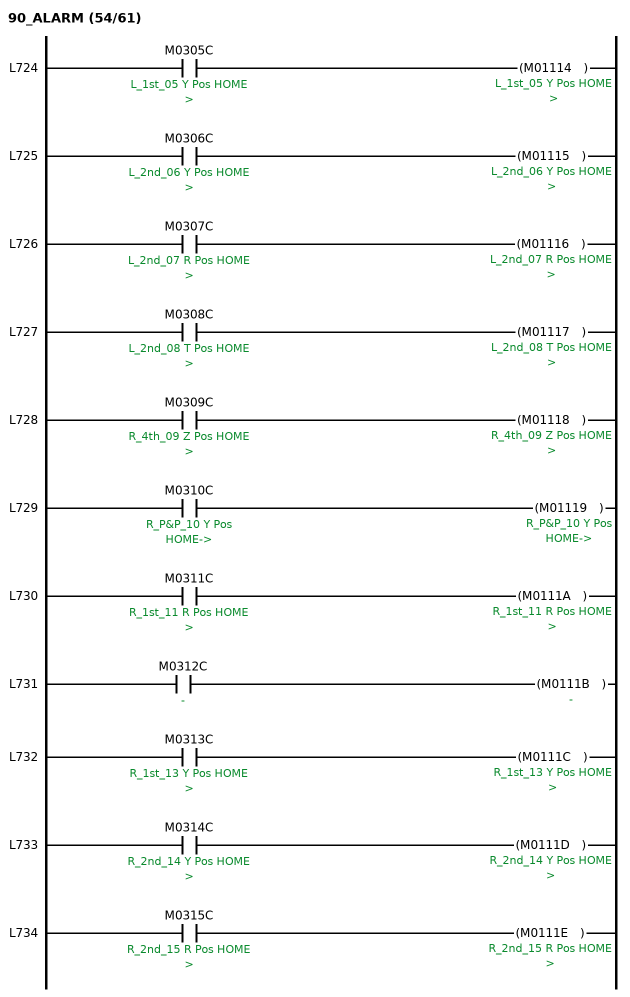
; L724
LOAD      M0305C	// L_1st_05 Y Pos HOME >
OUT       M01114	// L_1st_05 Y Pos HOME >
; L725
LOAD      M0306C	// L_2nd_06 Y Pos HOME >
OUT       M01115	// L_2nd_06 Y Pos HOME >
; L726
LOAD      M0307C	// L_2nd_07 R Pos HOME >
OUT       M01116	// L_2nd_07 R Pos HOME >
; L727
LOAD      M0308C	// L_2nd_08 T Pos HOME >
OUT       M01117	// L_2nd_08 T Pos HOME >
; L728
LOAD      M0309C	// R_4th_09 Z Pos HOME >
OUT       M01118	// R_4th_09 Z Pos HOME >
; L729
LOAD      M0310C	// R_P&P_10 Y Pos HOME->
OUT       M01119	// R_P&P_10 Y Pos HOME->
; L730
LOAD      M0311C	// R_1st_11 R Pos HOME >
OUT       M0111A	// R_1st_11 R Pos HOME >
; L731
LOAD      M0312C	// -
OUT       M0111B	// -
; L732
LOAD      M0313C	// R_1st_13 Y Pos HOME >
OUT       M0111C	// R_1st_13 Y Pos HOME >
; L733
LOAD      M0314C	// R_2nd_14 Y Pos HOME >
OUT       M0111D	// R_2nd_14 Y Pos HOME >
; L734
LOAD      M0315C	// R_2nd_15 R Pos HOME >
OUT       M0111E	// R_2nd_15 R Pos HOME >

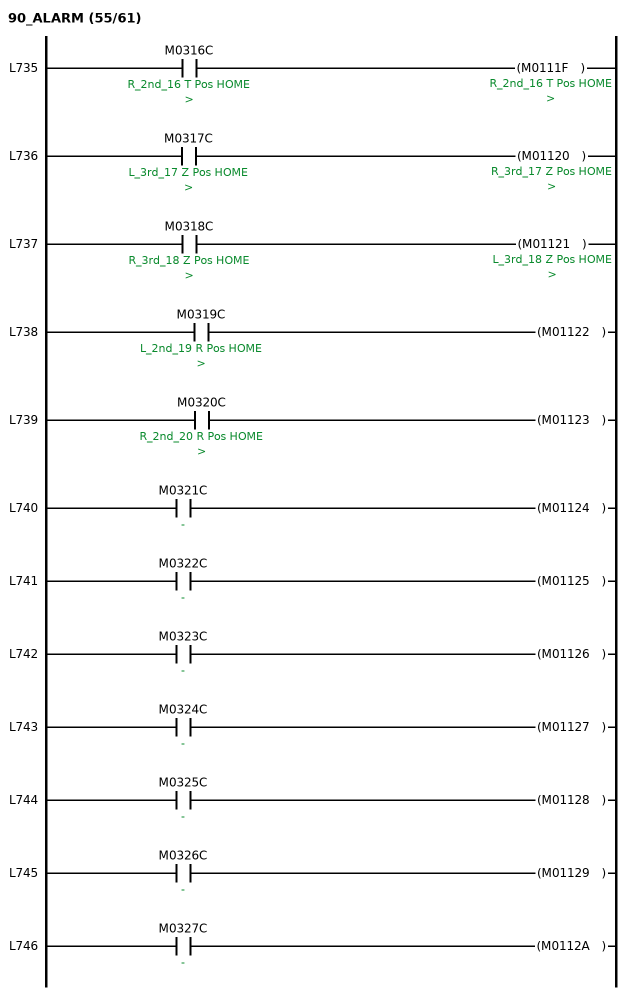
; L735
LOAD      M0316C	// R_2nd_16 T Pos HOME >
OUT       M0111F	// R_2nd_16 T Pos HOME >
; L736
LOAD      M0317C	// L_3rd_17 Z Pos HOME >
OUT       M01120	// R_3rd_17 Z Pos HOME >
; L737
LOAD      M0318C	// R_3rd_18 Z Pos HOME >
OUT       M01121	// L_3rd_18 Z Pos HOME >
; L738
LOAD      M0319C	// L_2nd_19 R Pos HOME >
OUT       M01122
; L739
LOAD      M0320C	// R_2nd_20 R Pos HOME >
OUT       M01123
; L740
LOAD      M0321C	// -
OUT       M01124
; L741
LOAD      M0322C	// -
OUT       M01125
; L742
LOAD      M0323C	// -
OUT       M01126
; L743
LOAD      M0324C	// -
OUT       M01127
; L744
LOAD      M0325C	// -
OUT       M01128
; L745
LOAD      M0326C	// -
OUT       M01129
; L746
LOAD      M0327C	// -
OUT       M0112A

